// TIA Portal project "LLCCA_PID" (V19)
// LCC Automation AB / (c)Copyright 2024
// Released under the MIT License

(* hardware
DEVICE "LLCCA_PID_HMI"  TP1200 Comfort
   slot 0: "LLCCA_PID_HMI"  TP1200 Comfort  6AV2 124-0MC01-0AX0  17.0.0.0
   slot 1: "HMI_RT_1"  TP1200 Comfort  6AV2 124-0MC01-0AX0  17.0.0.0
   slot 5: "LLCCA_PID_HMI.IE_CP_1"  PROFINET Interface  17.0.0.0
      slot 1: "PROFINET Interface_1"  PROFINET Interface
         slot 1: "Port_1"  Port
         slot 2: "Port_2"  Port
   slot 7: "LLCCA_PID_HMI.MPI/DP_CP_1"  MPI/DP Interface  17.0.0.0
DEVICE "ET 200SP station_1"  ET 200SP-Station
   slot 0: "Rack_0"  Rack  6ES5 710-8MAx1
   slot 1: "LLCCA_PID_PLC"  CPU 1510SP-1 PN  6ES7 510-1DK03-0AB0  V3.1
      slot 32768: "PROFINET interface_1"  X1
         slot 32771: "Port_3"  X1 P3
   slot 2: "Server module_1"  Server module  6ES7 193-6PA00-0AA0  V1.2
      slot 1: "Server module_1"  Server module
   slot 127: "BA 2xRJ45"  BA 2xRJ45  6ES7 193-6AR00-0AA0  V0.0
      slot 32769: "Port_1"  X1 P1  6ES7 193-6AR00-0AA0
      slot 32770: "Port_2"  X1 P2  6ES7 193-6AR00-0AA0
*)

// ===== PLC "LLCCA_PID_PLC"  CPU 1510SP-1 PN =====

DATA_BLOCK "LLCCA_PvSim_LLCCA_PID_DB"   // DB1
{ S7_Optimized_Access := 'TRUE' }
VERSION : 0.1
// stored: InstanceOfName LLCCA_PvSim
"LLCCA_PvSim"
BEGIN
END_DATA_BLOCK

DATA_BLOCK "LLCCA_PID_DB"   // DB2
{ S7_Optimized_Access := 'TRUE' }
AUTHOR : Jacob Holmdahl
VERSION : 0.0
// stored: InstanceOfName LLCCA_PID
"LLCCA_PID"
BEGIN
END_DATA_BLOCK

DATA_BLOCK "LLCCA_PvSim_PID_C_DB"   // DB3
{ S7_Optimized_Access := 'TRUE' }
VERSION : 0.1
// stored: InstanceOfName LLCCA_PvSim
"LLCCA_PvSim"
BEGIN
END_DATA_BLOCK

DATA_BLOCK "RUN_DB"   // DB5
{ S7_Optimized_Access := 'TRUE' }
VERSION : 0.1
// stored: InstanceOfName RUN
"RUN"
BEGIN
END_DATA_BLOCK

DATA_BLOCK "LLCCA_ErrAcc_DB_LLCCA_PID"   // DB10
{ S7_Optimized_Access := 'TRUE' }
VERSION : 0.1
// stored: InstanceOfName LLCCA_ErrAcc
"LLCCA_ErrAcc"
BEGIN
END_DATA_BLOCK

DATA_BLOCK "LLCCA_ErrAcc_DB_PID_C"   // DB11
{ S7_Optimized_Access := 'TRUE' }
VERSION : 0.1
// stored: InstanceOfName LLCCA_ErrAcc
"LLCCA_ErrAcc"
BEGIN
END_DATA_BLOCK

FUNCTION_BLOCK "RUN"   // FB1, FBD
{ S7_Optimized_Access := 'TRUE' }
AUTHOR : Jacob Holmdahl
VERSION : 0.0
   VAR_INPUT
      setpoint : Real;
   END_VAR
   VAR_IN_OUT
      resetAll : Bool;
      resetPvSim : Bool;
      resetPID : Bool;
      resetAccErr : Bool;
   END_VAR
   VAR
      statSetpoint : Real;
   END_VAR
   VAR_TEMP
      tempPv_LCCA_PID : Real;
      tempPv_PID_C : Real;
      tempResetPvSim : Bool;
      tempResetPID : Bool;
      tempResetAccErr : Bool;
   END_VAR
BEGIN

REGION Network 1 (SCL)
   IF #setpoint <> #statSetpoint THEN
     "LLCCA_PID_DB".Setpoint := #setpoint;
     "PID_Compact_1".Setpoint := #setpoint;
     #statSetpoint := #setpoint;
     #resetAccErr := TRUE;
   END_IF;
END_REGION

REGION Network 2
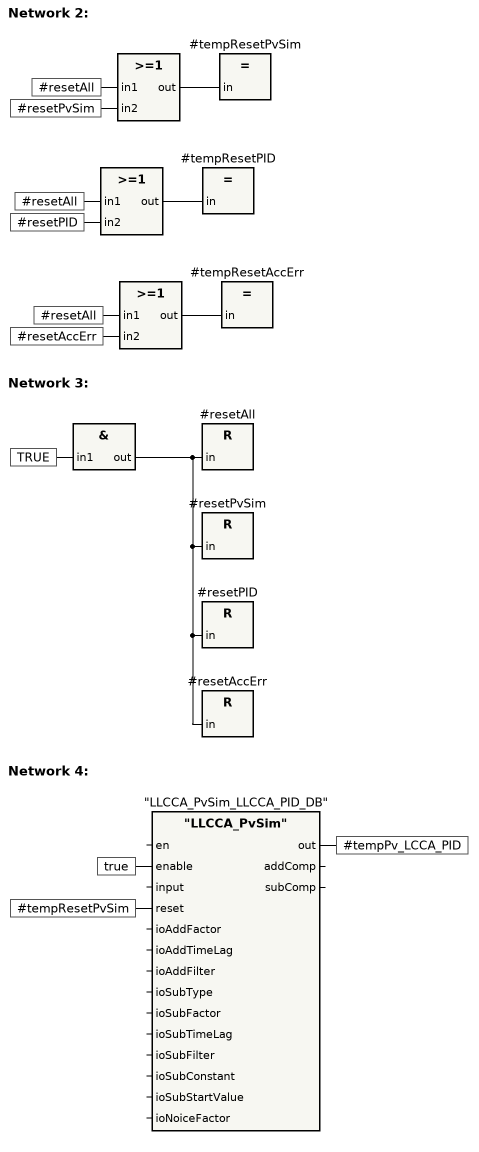
   #tempResetPvSim := #resetAll OR #resetPvSim;
   #tempResetPID := #resetAll OR #resetPID;
   #tempResetAccErr := #resetAll OR #resetAccErr;
END_REGION

REGION Network 3
   IF TRUE THEN
       #resetAll := FALSE;
       #resetPvSim := FALSE;
       #resetPID := FALSE;
       #resetAccErr := FALSE;
   END_IF;
END_REGION

REGION Network 4
   "LLCCA_PvSim_LLCCA_PID_DB"(enable := true, reset := #tempResetPvSim, out => #tempPv_LCCA_PID);   // "LLCCA_PvSim"
END_REGION

REGION Network 5
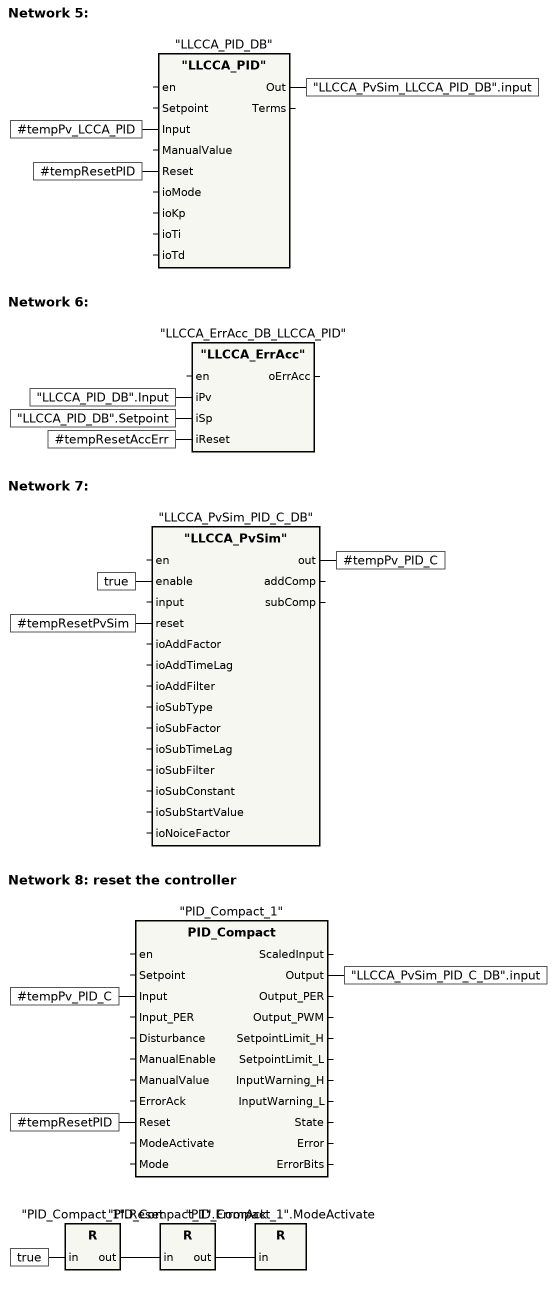
   "LLCCA_PID_DB"(Input := #tempPv_LCCA_PID, Reset := #tempResetPID, Out => "LLCCA_PvSim_LLCCA_PID_DB".input);   // "LLCCA_PID"
END_REGION

REGION Network 6
   "LLCCA_ErrAcc_DB_LLCCA_PID"(iPv := "LLCCA_PID_DB".Input,   // "LLCCA_ErrAcc"
                           iSp := "LLCCA_PID_DB".Setpoint,
                           iReset := #tempResetAccErr);
END_REGION

REGION Network 7
   "LLCCA_PvSim_PID_C_DB"(enable := true, reset := #tempResetPvSim, out => #tempPv_PID_C);   // "LLCCA_PvSim"
END_REGION

REGION Network 8: reset the controller
   "PID_Compact_1"(Input := #tempPv_PID_C, Reset := #tempResetPID, Output => "LLCCA_PvSim_PID_C_DB".input);   // PID_Compact
   IF true THEN
       "PID_Compact_1".Reset := FALSE;
       "PID_Compact_1".ErrorAck := FALSE;
       "PID_Compact_1".ModeActivate := FALSE;
   END_IF;
END_REGION

REGION Network 9
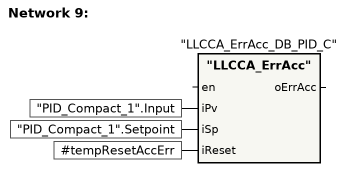
   "LLCCA_ErrAcc_DB_PID_C"(iPv := "PID_Compact_1".Input,   // "LLCCA_ErrAcc"
                           iSp := "PID_Compact_1".Setpoint,
                           iReset := #tempResetAccErr);
END_REGION
END_FUNCTION_BLOCK

FUNCTION_BLOCK "LLCCA_PID"   // FB3, SCL
TITLE = LLCCA_PID
{ S7_Optimized_Access := 'TRUE' }
AUTHOR : Jacob Holmdahl
FAMILY : LLCCA
VERSION : 0.0
// LCC Automation AB / (c)Copyright 2024
// Released under the MIT License
   VAR_INPUT
      Setpoint : Real;   // controller setpoint
      Input : Real;   // current value from the process
      ManualValue : Real;   // manual value
      Reset : Bool;   // reset i term and all filters
   END_VAR
   VAR_OUTPUT
      Out : Real;   // output value
      Terms : Struct   // controller terms
         p : Real;   // proportional term
         i : Real;   // integral term
         d : Real;   // derivative term
      END_STRUCT;
   END_VAR
   VAR_IN_OUT
      ioMode : USInt;   // current mode of operation (0-Inactive, 1-Step tuning, 2-Reserved, 3-Automatic, 4-Manual)
      ioKp : Real := 1.0;   // proportional gain
      ioTi : Real := 3.0;   // integral action time [s]
      ioTd : Real := 0.0;   // derivative action time [s]
   END_VAR
   VAR
      statOut : Real;
   END_VAR
   VAR RETAIN
      statAdvanced : Struct
         outMax : Real := 100.0;   // output value max
         outMin : Real;   // output value min
         inputFilter : Real := 0.1;   // input value filter time [s]
         derivateFilter : Real := 2.0;   // derivative filter time [s]
         tuningRule : USInt;   // 0:CHR 0% 1:0:CHR 20% 11:ZN fast 12:ZN normal 13:ZN slow
      END_STRUCT;
   END_VAR
   VAR
      statStepTuning : Struct
         state : USInt;
         stateInflection : USInt;
         t : Real;   // time
         find_u_max : Real;   // input max
         find_u_min : Real;   // input min
         calc_u_dev : Real;   // input deviation
         calc_u_start : Real;   // input start value
         find_y_start : Real;   // output start value
         find_k_inflection : Real;   // inflection point slope
         find_u_inflection : Real;   // inflection point input
         find_t_inflection : Real;   // inflection point time
         calc_m : Real;   // liniar equation
         calc_dy : Real;   // delta output
         calc_L : Real;   // apparent dead time
         calc_A : Real;
         calc_Kc : Real;
         calc_Ti : Real;
         calc_Td : Real;
      END_STRUCT;
      statErr : Real;
      statRuntime : LReal;
      statIntegralMax : Real;
      statIntegralMin : Real;
      statIntegralSum : Real;
      statMedianFilter : "LLCCA_MedianFilter";
      statFilterPT1 : Filter_PT1;
      "statFilterDT1_du/dt" : Filter_DT1;
      "statFilterDT1_d2u/dt2" : Filter_DT1;
      statMode : USInt;
      statModePrev : USInt;
   END_VAR
   VAR_TEMP
      temp_uM : Real;   // input with median filter
      temp_uF : Real;   // input with PT1 filter
      temp_dt : Real;   // delta time of the controller
      "temp_du/dt" : Real;   // first order derivative
      "temp_d2u/dt2" : Real;   // second order derivative
      temp_out : Real;
   END_VAR
BEGIN
   REGION Header
       //
       //================================================================================== 
       // LCC Automation AB / (c)Copyright 2024
       // Released under the MIT License
       //---------------------------------------------------------------------------------- 
       // Title:            LLCCA_PID
       // Comment/Function: PID Controller with step tuning
       // Library/Family:   LLCCA (Library LCC Automation AB)
       // Author:           Jacob Holmdahl / jacob.holmdahl@lcc.se
       // Target System:    CPU 1510SP-1
       // Engineering:      TIA Portal 19 update 3
       // Restrictions:     none
       // Requirements:     PLC (S7-1200 / S7-1500)
       //---------------------------------------------------------------------------------- 
       // Change log table: 
       // Version     | Date       | Author           | Changes applied
       //-------------|------------|------------------|------------------------------------ 
       // 000.002.000 | 2024-10-22 | Jacob Holmdahl   | PID with integral anti windup
       // 000.003.000 | 2024-11-10 | Jacob Holmdahl   | CHR and ZN step tuning
       // 000.003.001 | 2024-11-27 | Jacob Holmdahl   | First development release
       //==================================================================================
       //
       // Known issues
       // The step tuning only works if the process (input) is very stable.
       // An abort mechanism is needed to stop tuning if the process is or becomes unstable.
       //
       // Information
       // The terminology of some variables and functions is taken from the Siemens PID_Compact
       // controller.
       // 
   END_REGION

   REGION Save previous mode

       // one cycle mode change 
       IF #ioMode <> #statMode THEN
           #statModePrev := #statMode;
           #statMode := #ioMode;

           // init step tuning
           IF #statMode = 1 THEN
               #statStepTuning.state := 0;
               #statStepTuning.stateInflection := 0;
           END_IF;

       END_IF;

   END_REGION

   REGION Delta time
       // calculate the time from previous call = controller cycle time
       #temp_dt := LREAL_TO_REAL(RUNTIME(#statRuntime));
   END_REGION

   REGION Filter and derivatives

       // derivate filter min
       IF #statAdvanced.derivateFilter < 0.1 THEN
           #statAdvanced.derivateFilter := 0.1;
       END_IF;

       // filter setpoints
       #statFilterPT1.Lag := #statAdvanced.inputFilter;
       #"statFilterDT1_du/dt".Lag := #statAdvanced.derivateFilter;
       #"statFilterDT1_d2u/dt2".Lag := #statAdvanced.derivateFilter;

       // input value median filter
       #statMedianFilter(iVal := #Input,
                         iReset := #Reset,
                         oVal => #temp_uM);

       // reset all filters
       IF #Reset THEN
           #statFilterPT1.SubstituteOutput := #Input;
           #"statFilterDT1_du/dt".SubstituteOutput := 0.0;
           #"statFilterDT1_d2u/dt2".SubstituteOutput := 0.0;
       END_IF;

       // input value filter PT1
       #statFilterPT1(Input := #temp_uM,
                      Reset := #Reset,
                      Output => #temp_uF);

       // first order derivative
       // derivate filter DT1
       // returns the slope
       #"statFilterDT1_du/dt"(Input := #temp_uF,
                        Reset := #Reset,
                        Output => #"temp_du/dt");

       // second order derivative
       // derivate filter DT1 of the first derivate filter DT1
       // returns the acceleration of the slope
       #"statFilterDT1_d2u/dt2"(Input := #"temp_du/dt",
                        Reset := #Reset,
                        Output => #"temp_d2u/dt2");

   END_REGION

   REGION Modes

       CASE #statMode OF
           0:  // Inactive
               REGION Inactive
                   #statOut := 0.0;
               END_REGION

           1:  // Step tuning

               // The step tuning is designed to work with a FOPDT process model
               // FOPDT stands for First Order Plus Dead Time
               // First Order: This refers to a system that responds to a change in input with a gradual, exponential approach to a new steady state.
               // Dead Time: This represents a delay between when you make a change to the input and when you see any effect on the output. 

               REGION Step tuning

                   CASE #statStepTuning.state OF
                       0:

                           REGION Initialize tuning

                               // init tuning variables
                               #statStepTuning.find_u_max := #temp_uF;
                               #statStepTuning.find_u_min := #temp_uF;
                               #statStepTuning.calc_u_dev := 0.0;
                               #statStepTuning.calc_u_start := 0.0;
                               #statStepTuning.find_k_inflection := 0.0;
                               #statStepTuning.find_u_inflection := 0.0;
                               #statStepTuning.find_t_inflection := 0.0;
                               #statStepTuning.calc_m := 0.0;
                               #statStepTuning.calc_L := 0.0;
                               #statStepTuning.calc_Kc := 0.0;
                               #statStepTuning.calc_Ti := 0.0;
                               #statStepTuning.calc_Td := 0.0;
                               #statStepTuning.t := 5.0;

                               // transition
                               #statStepTuning.state := 1;

                           END_REGION

                       1:

                           REGION Calculate the standard deviation

                               // find min and max input
                               IF #temp_uF > #statStepTuning.find_u_max THEN
                                   #statStepTuning.find_u_max := #temp_uF;
                               END_IF;
                               IF #temp_uF < #statStepTuning.find_u_min THEN
                                   #statStepTuning.find_u_min := #temp_uF;
                               END_IF;

                               // calculate the standard deviation
                               #statStepTuning.calc_u_dev := #statStepTuning.find_u_max - #statStepTuning.find_u_min;

                               // transition
                               // timer run out / calculate starting point
                               IF #statStepTuning.t <= 0.0 THEN
                                   #statStepTuning.t := 0.0;

                                   // adjust derivate filter to coresponting deviation
                                   #statAdvanced.derivateFilter := #statStepTuning.calc_u_dev * 40.0;
                                   #statAdvanced.derivateFilter := #statStepTuning.calc_u_dev * 40.0;

                                   // save starting point
                                   #statStepTuning.calc_u_start := #statStepTuning.find_u_min + #statStepTuning.calc_u_dev / 2;
                                   #statStepTuning.find_k_inflection := #"temp_du/dt"; // save slope

                                   // save start output
                                   #statStepTuning.find_y_start := #statOut;

                                   // increase output to make a step
                                   #statOut := #statAdvanced.outMax;

                                   // change state
                                   #statStepTuning.state := 2;
                               ELSE
                                   // decrease step timer
                                   #statStepTuning.t := #statStepTuning.t - #temp_dt;
                               END_IF;

                           END_REGION

                       2:

                           REGION Find the point of inflection

                               // terminology
                               // L = Deadtime ( Can also be called τ in some documantations )
                               // T = apparent time constant
                               // y = output

                               // linear equation
                               // u = kt + m ( u=pv , t=time )
                               // k = u2-u1 / t2-t1 = du / dt

                               // finding inflection point = k
                               IF #"temp_du/dt" > #statStepTuning.find_k_inflection THEN
                                   #statStepTuning.find_k_inflection := #"temp_du/dt";
                                   #statStepTuning.find_u_inflection := #temp_uF;
                                   #statStepTuning.find_t_inflection := #statStepTuning.t;
                               END_IF;

                               // calculate m from inflection point
                               // u=kt+m => m=u-kt 
                               #statStepTuning.calc_m := #statStepTuning.find_u_inflection - (#statStepTuning.find_k_inflection * #statStepTuning.find_t_inflection);

                               // calculate L, the "apparent dead time" with u=kt+m => t=u-m/k at the staring level.
                               #statStepTuning.calc_L := (#statStepTuning.calc_u_start - #statStepTuning.calc_m) / #statStepTuning.find_k_inflection;

                               // calculate delta y (delta output)
                               #statStepTuning.calc_dy := #statAdvanced.outMax - #statStepTuning.find_y_start;

                               // A = approximation of KL/T
                               #statStepTuning.calc_A := #statStepTuning.calc_u_start - #statStepTuning.calc_m;

                               // increase timer / tuning time t
                               #statStepTuning.t := #statStepTuning.t + #temp_dt;

                               // start tuning
                               IF #statStepTuning.stateInflection = 0 AND #"statFilterDT1_du/dt".Output > 0.1 THEN
                                   #statStepTuning.stateInflection := 1;
                               END_IF;

                               // end tuning
                               IF #statStepTuning.stateInflection = 1 AND #"statFilterDT1_d2u/dt2".Output < 0.0 THEN
                                   #statStepTuning.stateInflection := 2;
                               END_IF;

                               // transition to "Tuning successful"
                               IF #statStepTuning.stateInflection = 2 THEN
                                   #statStepTuning.state := 3;
                               END_IF;



                               CASE #statAdvanced.tuningRule OF

                                   0: // Chien–Hrones–Reswick - tuning for disturbance rejection - with 0% overshot
                                       #statStepTuning.calc_Kc := (0.95 * #statStepTuning.calc_dy) / #statStepTuning.calc_A;
                                       #statStepTuning.calc_Ti := 2.40 * #statStepTuning.calc_L;
                                       #statStepTuning.calc_Td := 0.42 * #statStepTuning.calc_L;
                                   1: // Chien–Hrones–Reswick - tuning for disturbance rejection - with 20% overshot
                                       #statStepTuning.calc_Kc := (1.20 * #statStepTuning.calc_dy) / #statStepTuning.calc_A;
                                       #statStepTuning.calc_Ti := 2.00 * #statStepTuning.calc_L;
                                       #statStepTuning.calc_Td := 0.42 * #statStepTuning.calc_L;
                                   11:  // Ziegler-Nichols - Fast Performance
                                       #statStepTuning.calc_Kc := (1.20 * #statStepTuning.calc_dy) / #statStepTuning.calc_A;
                                       #statStepTuning.calc_Ti := 2.00 * #statStepTuning.calc_L;
                                       #statStepTuning.calc_Td := 0.50 * #statStepTuning.calc_L;
                                   12:  // Ziegler-Nichols - Normal Performance
                                       #statStepTuning.calc_Kc := (0.53 * #statStepTuning.calc_dy) / #statStepTuning.calc_A;
                                       #statStepTuning.calc_Ti := 4.00 * #statStepTuning.calc_L;
                                       #statStepTuning.calc_Td := 0.80 * #statStepTuning.calc_L;
                                   13:  // Ziegler-Nichols - Slow Performance
                                       #statStepTuning.calc_Kc := (0.32 * #statStepTuning.calc_dy) / #statStepTuning.calc_A;
                                       #statStepTuning.calc_Ti := 4.00 * #statStepTuning.calc_L;
                                       #statStepTuning.calc_Td := 0.80 * #statStepTuning.calc_L;

                                   ELSE  // Statement section ELSE

                                       #statAdvanced.tuningRule := 0;

                               END_CASE;

                           END_REGION


                       3:

                           REGION Tuning successful

                               // set new tuning parameters
                               #ioKp := #statStepTuning.calc_Kc;
                               #ioTi := #statStepTuning.calc_Ti;
                               #ioTd := #statStepTuning.calc_Td;

                               // return to previous mode
                               #ioMode := #statModePrev;

                           END_REGION

                       4:

                           REGION Tuning not successful

                               // return to previous mode
                               #ioMode := #statModePrev;

                           END_REGION

                       ELSE  // error
                           ;
                   END_CASE;

               END_REGION

           2:  // Reserved for future mode
               REGION Reserved for future mode

                   // prohibited mode - inactivate controller
                   #ioMode := 0;

               END_REGION

           3:  // Automatic
               REGION Automatic

                   // error calculation
                   #statErr := #Setpoint - #temp_uF;

                   REGION PID terms

                       // proprtional gain term
                       #Terms.p := #ioKp * #statErr;

                       // derivate term
                       #Terms.d := - #ioKp * #ioTd * #"temp_du/dt";

                       // integral sum
                       #statIntegralSum := #statIntegralSum + ((#statErr * #temp_dt) / #ioTi);

                       // integral reset
                       IF #Reset THEN
                           #statIntegralSum := 0.0;
                       END_IF;

                       REGION Anti-integral windup

                           // integral max and min
                           #statIntegralMax := (#statAdvanced.outMax / #ioKp) - (#Terms.d / #ioKp) - #statErr;
                           #statIntegralMin := (#statAdvanced.outMin / #ioKp) - (#Terms.d / #ioKp) - #statErr;

                           // integral max with positive error
                           IF #statIntegralSum >= #statIntegralMax AND #statErr > 0.0 THEN
                               #statIntegralSum := #statIntegralMax;
                           END_IF;

                           // integral mmin with negative error
                           IF #statIntegralSum <= #statIntegralMin AND #statErr < 0.0 THEN
                               #statIntegralSum := #statIntegralMin;
                           END_IF;
                       END_REGION

                       // integral term
                       IF #ioTi > 0.0 THEN
                           #Terms.i := #ioKp * #statIntegralSum;
                       ELSE
                           #ioTi := 0.0;
                           #Terms.i := 0.0;
                       END_IF;

                   END_REGION

                   REGION Output

                       // calculate temporary output
                       #temp_out := #Terms.p + #Terms.i + #Terms.d;

                       // min and max limit
                       IF #temp_out < #statAdvanced.outMin THEN
                           #temp_out := #statAdvanced.outMin;
                       ELSIF #temp_out > #statAdvanced.outMax THEN
                           #temp_out := #statAdvanced.outMax;
                       END_IF;

                       // set output vaiable
                       #statOut := #temp_out;

                   END_REGION

               END_REGION

           4:  // Manual
               REGION Manual

                   // set manual output
                   #statOut := #ManualValue;

               END_REGION

           ELSE  // prohibited mode - inactivate controller

               #ioMode := 0;

       END_CASE;

   END_REGION

   REGION Output value
       #Out := #statOut;
   END_REGION
END_FUNCTION_BLOCK

FUNCTION_BLOCK "LLCCA_PvSim"   // FB19, SCL
TITLE = LLCCA_PvSim
{ S7_Optimized_Access := 'TRUE' }
AUTHOR : Jacob Holmdahl
FAMILY : LLCCA
VERSION : 0.0
// LCC Automation AB / (c)Copyright 2024
// Released under the MIT License
   VAR_INPUT
      enable : Bool;   // enable simulation
      input : Real;   // input (Output from PID) [%]
      reset : Bool;   // reset
   END_VAR
   VAR_OUTPUT
      out : Real;   // simulated process value [unit]
      addComp : Real;   // additive component [unit/min]
      subComp : Real;   // subtracting component [unit/min]
   END_VAR
   VAR_IN_OUT
      ioAddFactor : Real := 1.0;   // additive component factor ( addComp := input * addFactor ; 100% * 0.01 = 1 unit/min )
      ioAddTimeLag : USInt := 1;   // additive component time lag [s]
      ioAddFilter : Real := 5.0;   // additive component filter [s]
      ioSubType : USInt;   // 0:start val proportial 1:constant
      ioSubFactor : Real := 1.0;   // subtracting component factor ( subComp := ( out - subStartVal ) * subFactor ; sub (120 unit - 20 unit *0.01 = 1 unit/min)
      ioSubTimeLag : USInt;   // subtracting component time lag [s]
      ioSubFilter : Real;   // subtracting component filter [s]
      ioSubConstant : Real := 20.0;   // substracting constant
      ioSubStartValue : Real := 20.0;   // subtracting component start value [unit]
      ioNoiceFactor : Real := 0.1;   // random noice factor of simulated process value
   END_VAR
   VAR
      statOut : Real;
      statRuntimeMem : LReal;
      statAddTimeLag : "LLCCA_TimeLag";
      statAddFilter_PT1 : Filter_PT1;
      statSubTimeLag : "LLCCA_TimeLag";
      statSubFilter_PT1 : Filter_PT1;
   END_VAR
   VAR_TEMP
      tempDeltaTime : LReal;
      tempAdd : Real;
      tempSub : Real;
      tempRndError : Bool;
      tempRndStatus : Word;
      tempRndStatusSub : Word;
   END_VAR
BEGIN
   REGION Description header 
       //================================================================================== 
       // LCC Automation AB / (c)Copyright 2024
       // Released under the MIT License
       //---------------------------------------------------------------------------------- 
       // Title:            LLCCA_PvSim
       // Comment/Function: Process value simulator
       // Library/Family:   LLCCA (Library LCC Automation AB)
       // Author:           Jacob Holmdahl / jacob.holmdahl@lcc.se
       // Target System:    CPU 1510SP-1
       // Engineering:      TIA Portal 19 update 3
       // Restrictions:     none
       // Requirements:     PLC (S7-1200 / S7-1500)
       //---------------------------------------------------------------------------------- 
       // Change log table: 
       // Version     | Date       | Author           | Changes applied
       //-------------|------------|------------------|------------------------------------ 
       // 001.000.000 | 2024-11-27 | Jacob Holmdahl   | First release
       //==================================================================================
   END_REGION

   REGION delta time
       #tempDeltaTime := RUNTIME(#statRuntimeMem);
   END_REGION

   REGION reset

     IF #reset OR NOT #enable THEN
       #statOut := #ioSubStartValue;
   END_IF;

   END_REGION

   REGION limits

     IF #ioAddFilter < 0.00 THEN
       #ioAddFilter := 0.00;
     END_IF;

     IF #ioSubFilter < 0.00 THEN
       #ioSubFilter := 0.00;
     END_IF;

   END_REGION

   REGION add component

     #tempAdd := #input / 1.0;

     IF ENO THEN
         #tempAdd := #input * #ioAddFactor;
     ELSE
       #tempAdd := 0.0;
     END_IF;

   END_REGION

   REGION add timeLag

     #statAddTimeLag(in      := #tempAdd,
                     reset   := #reset,
                     timeLag := #ioAddTimeLag);

   END_REGION

   REGION add filter

     IF #ioAddFilter > 0.01 THEN
       #statAddFilter_PT1.Lag := #ioAddFilter;

       #statAddFilter_PT1(Input            := #statAddTimeLag.out,
                          SubstituteOutput := #statAddTimeLag.out,
                          Reset            := #reset,
                          Output           => #tempAdd);
     ELSE
       #tempAdd := #statAddTimeLag.out;
     END_IF;

     #addComp := #tempAdd;

   END_REGION

   REGION addition

     #statOut := #statOut + ((#tempAdd * LREAL_TO_REAL(#tempDeltaTime)) / 60.0);

   END_REGION

   REGION sub component

     IF #ioSubType = 0 THEN

       #tempSub := (#statOut - #ioSubStartValue) * #ioSubFactor;

     ELSIF #ioSubType = 1 THEN

       IF #statOut > #ioSubStartValue THEN
         #tempSub := #ioSubConstant * #ioSubFactor;
       ELSE
         #statOut := #ioSubStartValue;
       END_IF;

     ELSE
       #ioSubType := 0;
     END_IF;

   END_REGION

   REGION sub timeLag

     #statSubTimeLag(in      := #tempSub,
                     reset   := #reset,
                     timeLag := #ioSubTimeLag);

   END_REGION

   REGION sub filter

     IF #ioSubFilter > 0.01 THEN
       #statSubFilter_PT1.Lag := #ioSubFilter;

       #statSubFilter_PT1(Input            := #statSubTimeLag.out,
                          SubstituteOutput := #statSubTimeLag.out,
                          Reset            := #reset,
                          Output           => #tempSub);
     ELSE
       #tempSub := #statSubTimeLag.out;
     END_IF;

     #subComp := #tempSub;

   END_REGION

   REGION substraction

     #statOut := #statOut - (#tempSub * LREAL_TO_REAL(#tempDeltaTime) / 60.0);

   END_REGION

   REGION output and noice
     #out := #statOut - (0.5 * #ioNoiceFactor) + #ioNoiceFactor * "LGF_Random_Real"(error => #tempRndError, status => #tempRndStatus, subfunctionStatus => #tempRndStatusSub);
   END_REGION
END_FUNCTION_BLOCK

ORGANIZATION_BLOCK "Main"   // OB1, FBD, ProgramCycle
TITLE = "Main Program Sweep (Cycle)"
{ S7_Optimized_Access := 'TRUE' }
VERSION : 0.1
   VAR_INPUT
      Initial_Call : Bool;   // Initial call of this OB
      Remanence : Bool;   // =True, if remanent data are available
   END_VAR
BEGIN

REGION Network 1
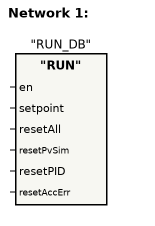
   "RUN_DB"();   // "RUN"
END_REGION
END_ORGANIZATION_BLOCK

// folder: LGF

FUNCTION "LGF_Random_Real" : Real   // FC10077, SCL
TITLE = LGF_Random_Real
{ S7_Optimized_Access := 'TRUE' }
AUTHOR : Siemens_Digital_Industries
FAMILY : LGF
NAME : LGF_Random_Real
// This function generates a random value with each call.  
// The random number has the data type Real in the range from 0.0 to 1.0.
// Diese Funktion generiert bei jedem Aufruf einen zufälligen Wert.  
// Die Zufallszahl hat den Datentyp Real und den Wertebereich von 0.0 bis 1.0.
   VAR_OUTPUT
      error : Bool;   // FALSE: No error TRUE: An error occurred during the execution of the FB / FALSE: Kein Fehler TRUE: Während der Ausführung des FB ist ein Fehler aufgetreten
      status : Word;   // 16#0000-16#7FFF: Status of the FB 16#8000-16#FFFF: Error identification (see following Table) / 16#0000-16#7FFF: Status des FB 16#8000-16#FFFF: Fehleridentifikation (siehe folgende Tabelle)
      subfunctionStatus : Word;   // Status or return value of called FB's, FC's and system blocks / Status oder Rückgabewert von aufgerufenen FB's / FC's und Systemfunktionen
   END_VAR
   VAR_TEMP
      tempTime : DTL;   // Temp memory for System time / Temp variable für System Zeit
      tempNanoSecondInDWord : DWord;   // Temp UDInt converted to DWord for access to individual bytes / Temp UDInt konvertiert nach Dword für den Zufriff per Slice auf die Bytes
      tempTimeStatus : Word;   // Temp status of the instruction `RD_SYS_T` / Temp Status der Systemfunktion `RD_SYS_T`
      tempRandomValue : DWord;   // Temp Random startvalue / Temp Zufallswert als Startwert
   END_VAR
   // Ret_Val : Random Real number between 0.0 and 1.0 / Zufallszahl vom Datentyp Real im Wertebereich von 0.0 bis 1.0
   VAR CONSTANT
      ZERO : Real;   // Zero / 0.0 - value in case of error / Null / 0.0 - Rückgabewert im Fehlerfall
      MAX_UDINT : UDInt := 4294967295 ;   // Maximum UDInt datatype / Maximalwert eines UDInt Datentype
      SUB_STATUS_NO_ERROR : Word := 16#0000;   // Status: sub function call ends without error / Status: Unterfunktionsaufruf ohne Fehler beendet
      STATUS_FINISHED_NO_ERROR : Word := 16#0000;   // Execution finished without errors / Abarbeitung ohne Fehler beendet
      ERR_RD_SYS_T : Word := 16#8600;   // Error in `RD_SYS_T` command - check `subFunctionStatus` code / Fehler in Anweisung `RD_SYS_T` - weitere infos in `subFunctionStatus`
   END_VAR
BEGIN
   REGION Block info header
     //=============================================================================
     // SIEMENS AG / (c)Copyright 2017
     //-----------------------------------------------------------------------------
     // Title:            LGF_Random_Real
     // Comment/Function: Generates a random real number between 0.0 and 1.0
     // Library/Family:   LGF(Library General Functions)
     // Author:           Siemens Digital Industry Support
     // Tested with:      S7-PLCSIM Advanced V2.0 SP1
     // Engineering:      TIA Portal V15 Update 2
     // Restrictions:     ENO disabled - error handling done by error and status
     // Requirements:     PLC (S7-1200 / S7-1500)
     //-------------------------------------------------------------------------------
     // Change log table:
     // Version  | Date       | Expert in charge       | Changes applied
     //----------|------------|------------------------|------------------------------
     // 01.00.00 27.01.2017  Siemens Industry Online Support
     //                      First released version
     // 01.00.01 17.08.2018  Siemens Industry Online Support
     //                      Upgrade: TIA V15 Update 2
     // 01.00.02 23.11.2018  Siemens Industry Online Support
     //                      Upgrade: TIA V15.1
     // 01.01.00 13.11.2019  Simatic Systems Support
     //                      Renamed from "LGF_RandomBasic" to "LGF_Random_Real"
     //                      Regions, comments and constants are added
     // 03.00.00 23.04.2020  Simatic Systems Support
     //                      Set version to V3.0.0, harmonize the version of the whole library
     // 03.00.01 04.02.2021  Simatic Systems Support
     //                      Insert documentation
     //=============================================================================
   END_REGION Block info header

   REGION DESCRIPTION
     (/*Note
   :    The status of called commands is output in `subFunctionStatus`. In this case, the output value in `status` indicates which command caused the error. In this case, refer to the TIA Portal Online Help section for information on the respective commands.

   The function generates random values in the range:  
   $ 0.0 ≤ ReturnVal ≤ 1.0 $.

   The random value is formed from the nanoseconds of the current system time of the CPU. The byte order of this value is inverted and then converted to a floating point.
   Hinweis
   :    In `subFunctionStatus` wird der Status von aufgerufenen Anweisungen ausgegeben. Der Ausgangswert in `status` gibt in diesem Fall an, welche Anweisung den Fehler verursacht hat. Holen Sie sich in diesem Fall die Informationen aus der TIA Portal Online Hilfe zu den jeweiligen Anweisungen.

   Die Funktion generiert zufällige Werte im Bereich:  
   $ 0.0 ≤ ReturnVal ≤ 1.0 $.

   Der Zufallswert wird aus den Nanosekunden der aktuellen Systemzeit der CPU gebildet. Dabei wird die Bytereihenfolge dieses Wertes invertiert und anschließend in eine Gleitkommazahl ungewandelt.*/)
   END_REGION DESCRIPTION

   REGION Validation
     // Read system time
     #tempTimeStatus := INT_TO_WORD(RD_SYS_T(#tempTime));

     // Check return variable for error
     IF (#tempTimeStatus <> #SUB_STATUS_NO_ERROR) THEN
       #error := true;
       #status := #ERR_RD_SYS_T;
       #subfunctionStatus := #tempTimeStatus;
       #LGF_Random_Real := #ZERO;
       RETURN;
     END_IF;
   END_REGION

   REGION Calculating random number
     // Converting to double word so individual bytes can be addressed
     #tempNanoSecondInDWord := UDINT_TO_DWORD(#tempTime.NANOSECOND);

     // Calculate a random-start-value depending on the time
     #tempRandomValue.%B3 := #tempNanoSecondInDWord.%B0;
     #tempRandomValue.%B2 := #tempNanoSecondInDWord.%B1;
     #tempRandomValue.%B1 := #tempNanoSecondInDWord.%B2;
     #tempRandomValue.%B0 := #tempNanoSecondInDWord.%B3;

     // Norm the calculated random number: 0.0 <= Random_Real <= 1.0
     #LGF_Random_Real := UDINT_TO_REAL(DWORD_TO_UDINT(#tempRandomValue)) / UDINT_TO_REAL(#MAX_UDINT);

     #error := false;
     #status := #STATUS_FINISHED_NO_ERROR;
     #subfunctionStatus := #SUB_STATUS_NO_ERROR;
     // ENO mechanism is not used
     ENO := TRUE;
   END_REGION
END_FUNCTION

// folder: SupportFunctions

FUNCTION_BLOCK "LLCCA_ErrAcc"   // FB2, SCL
TITLE = LLCCA_ErrAcc
{ S7_Optimized_Access := 'TRUE' }
AUTHOR : Jacob Holmdahl
FAMILY : LLCCA
VERSION : 0.1
// LCC Automation AB / (c)Copyright 2024
// Released under the MIT License
   VAR_INPUT
      iPv : Real;   // process value
      iSp : Real;   // setpoint
      iReset : Bool;   // reset
   END_VAR
   VAR_OUTPUT
      oErrAcc : LReal;   // error accumulator output
   END_VAR
   VAR
      statErrAcc : LReal;
      statRuntime : LReal;
   END_VAR
   VAR_TEMP
      tempDeltaTime : LReal;
   END_VAR
BEGIN
   REGION Description header 
       //================================================================================== 
       // LCC Automation AB / (c)Copyright 2024
       // Released under the MIT License
       //---------------------------------------------------------------------------------- 
       // Title:            LLCCA_ErrAcc
       // Comment/Function: Process value to setpoint error accumulator
       // Library/Family:   LLCCA (Library LCC Automation AB)
       // Author:           Jacob Holmdahl / jacob.holmdahl@lcc.se
       // Target System:    CPU 1510SP-1
       // Engineering:      TIA Portal 19 update 3
       // Restrictions:     none
       // Requirements:     PLC (S7-1200 / S7-1500)
       //---------------------------------------------------------------------------------- 
       // Change log table: 
       // Version     | Date       | Author           | Changes applied
       //-------------|------------|------------------|------------------------------------ 
       // 001.000.001 | 2024-11-27 | Jacob Holmdahl   | First release
       //==================================================================================
   END_REGION

   #tempDeltaTime := RUNTIME(#statRuntime);

   IF #iReset THEN
       #statErrAcc := 0.0;
   ELSE
       #statErrAcc := #statErrAcc + (ABS(#iSp - #iPv) * #tempDeltaTime);
   END_IF;

   // set output
   #oErrAcc := #statErrAcc;
END_FUNCTION_BLOCK

FUNCTION_BLOCK "LLCCA_MedianFilter"   // FB4, SCL
TITLE = LLCCA_MedianFilter
{ S7_Optimized_Access := 'TRUE' }
AUTHOR : Jacob Holmdahl
FAMILY : LLCCA
VERSION : 0.0
// LCC Automation AB / (c)Copyright 2024
// Released under the MIT License
   VAR_INPUT
      iVal : Real;   // input value
      iReset : Bool;   // reset
   END_VAR
   VAR_OUTPUT
      oVal : Real;   // output value
   END_VAR
   VAR
      statBuffer : Array[0..#UNITS] of Real;
   END_VAR
   VAR_TEMP
      findValue : Real;
      i : Int;
      j : Int;
      tempBuffer : Array[0..#UNITS] of Real;
   END_VAR
   VAR CONSTANT
      UNITS : Int := 31;
   END_VAR
BEGIN
   REGION Description header 
       //================================================================================== 
       // LCC Automation AB / (c)Copyright 2024
       // Released under the MIT License
       //---------------------------------------------------------------------------------- 
       // Title:            LLCCA_MedianFilter
       // Comment/Function: Median filter
       // Library/Family:   LLCCA (Library LCC Automation AB)
       // Author:           Jacob Holmdahl / jacob.holmdahl@lcc.se
       // Target System:    CPU 1510SP-1
       // Engineering:      TIA Portal 19 update 3
       // Restrictions:     none
       // Requirements:     PLC (S7-1200 / S7-1500)
       //---------------------------------------------------------------------------------- 
       // Change log table: 
       // Version     | Date       | Author           | Changes applied
       //-------------|------------|------------------|------------------------------------ 
       // 001.000.000 | 2024-11-27 | Jacob Holmdahl   | First release
       //==================================================================================
   END_REGION

   IF #iReset THEN

       // fill buffer with input val
       FOR #i := 0 TO #UNITS DO
           #statBuffer[#i] := #iVal;
       END_FOR;

       // output is set to input
       #oVal := #iVal;

   ELSE

       // move the static buffer one step
       // and fill the temp buffer
       FOR #i := #UNITS TO 1 BY -1 DO
           #statBuffer[#i] := #statBuffer[#i - 1];
           #tempBuffer[#i] := #statBuffer[#i];
       END_FOR;

       // save the actual value to the buffers
       #statBuffer[0] := #iVal;
       #tempBuffer[0] := #iVal;

       // sort the temp buffer
       FOR #i := 0 TO #UNITS DO
           FOR #j := 0 TO #UNITS - 1 DO
               IF #tempBuffer[#j] > #tempBuffer[#j + 1] THEN
                   #findValue := #tempBuffer[#j];
                   #tempBuffer[#j] := #tempBuffer[#j + 1];
                   #tempBuffer[#j + 1] := #findValue;
               END_IF;
           END_FOR;
       END_FOR;

       // set median val output
       #oVal := (#tempBuffer[#UNITS / 2] + #tempBuffer[#UNITS / 2 + 1]) / 2;

   END_IF;
END_FUNCTION_BLOCK

FUNCTION_BLOCK "LLCCA_TimeLag"   // FB18, SCL
TITLE = LLCCA_TimeLag
{ S7_Optimized_Access := 'TRUE' }
AUTHOR : Jacob Holmdahl
FAMILY : LLCCA
VERSION : 0.0
// LCC Automation AB / (c)Copyright 2024
// Released under the MIT License
   VAR_INPUT
      in : Real;   // input value
      init : Bool;   // time lag memory = in
      reset : Bool;   // time lag memory = 0.0
   END_VAR
   VAR_OUTPUT
      out : Real;   // output value
   END_VAR
   VAR_IN_OUT
      timeLag : USInt := 10;   // time lag [s]
   END_VAR
   VAR
      statRuntimeMem : LReal;
      statTimeLag : Array[0..#TIME_LAG_MAX] of Real;
      statTimer : LReal;
      statInit : Bool;
      statReset : Bool;
   END_VAR
   VAR_TEMP
      tempCycleTime : LReal;
      i : USInt;
   END_VAR
   VAR CONSTANT
      TIME_CYCLE : Real := 0.1;
      TIME_LAG_MAX : USInt := 250;
   END_VAR
BEGIN
   REGION Description header 
       //================================================================================== 
       // LCC Automation AB / (c)Copyright 2024
       // Released under the MIT License
       //---------------------------------------------------------------------------------- 
       // Title:            LLCCA_PID
       // Comment/Function: The output value is delayed by an adjustable time
       // Library/Family:   LLCCA (Library LCC Automation AB)
       // Author:           Jacob Holmdahl / jacob.holmdahl@lcc.se
       // Target System:    CPU 1510SP-1
       // Engineering:      TIA Portal 19 update 3
       // Restrictions:     none
       // Requirements:     PLC (S7-1200 / S7-1500)
       //---------------------------------------------------------------------------------- 
       // Change log table: 
       // Version     | Date       | Author           | Changes applied
       //-------------|------------|------------------|------------------------------------ 
       // 001.000.001 | 2024-11-27 | Jacob Holmdahl   | First release
       //==================================================================================
   END_REGION

   IF #timeLag > 0 THEN

     // run time lag code

     REGION cycleTime
       #tempCycleTime := RUNTIME(#statRuntimeMem);
     END_REGION
     //------------------------------------------------------------------------------------------
     REGION init

       IF #init AND NOT #statInit THEN
         #statInit := TRUE;
         #statTimer := #TIME_CYCLE;
         FOR #i := 0 TO #TIME_LAG_MAX DO
           #statTimeLag[#i] := #in;
         END_FOR;
       ELSIF NOT #init THEN
         #statInit := FALSE;
       END_IF;

     END_REGION
     //------------------------------------------------------------------------------------------
     REGION reset

       IF #reset AND NOT #statReset THEN
         #statReset := TRUE;
         #statTimer := #TIME_CYCLE;
         FOR #i := 0 TO #TIME_LAG_MAX DO
           #statTimeLag[#i] := 0.0;
         END_FOR;
       ELSIF NOT #reset THEN
         #statReset := FALSE;
       END_IF;

     END_REGION
     //------------------------------------------------------------------------------------------
     REGION limits

       // max
       IF #timeLag > #TIME_LAG_MAX/10 THEN
         #timeLag := #TIME_LAG_MAX/10;
       END_IF;

     END_REGION
     //------------------------------------------------------------------------------------------
     // decrease timer
     #statTimer := #statTimer - #tempCycleTime;

     // save value to memory
     IF #statTimer < 0.0 THEN
       #statTimer := #TIME_CYCLE;

       FOR #i := 0 TO #TIME_LAG_MAX-1 DO
         #statTimeLag[#TIME_LAG_MAX - #i] := #statTimeLag[#TIME_LAG_MAX - #i - 1];
       END_FOR;
       #statTimeLag[0] := #in;

     END_IF;

     // set output
     #out := #statTimeLag[#timeLag*10];

   ELSE
     // no time lag

     // set output
     #out := #in;

   END_IF;
END_FUNCTION_BLOCK

// ===== library types =====

// folder: LGF

FUNCTION "LGF_Description" : Void   // FC10087, SCL
TITLE = LGF_Description
{ S7_Optimized_Access := 'TRUE' }
AUTHOR : Siemens Industry Support
NAME : LGF_Description
// Block for the Libray description
BEGIN

   REGION INFO
     (/*title: Library of General Functions (LGF) for SIMATIC S7-1200 / S7-1500
   subTitle: STEP 7 Basic/Professional (TIA PORTAL)
   fileName: LGF
   siosId: 109479728
   link: https://support.industry.siemens.com/cs/ww/en/view/109479728
   classification:   
   # " " "Frei verwendbar" "Unrestricted" "Intern" "Restricted" "Vertraulich" "Confidential" "Streng vertraulich" "Strictly Confidential"
   title: Library of General Functions (LGF) für SIMATIC S7-1200 / S7-1500
   subTitle: STEP 7 Basic/Professional (TIA PORTAL)
   fileName: LGF
   siosId: 109479728
   link: https://support.industry.siemens.com/cs/ww/de/view/109479728
   classification:   
   # " " "Frei verwendbar" "Unrestricted" "Intern" "Restricted" "Vertraulich" "Confidential" "Streng vertraulich" "Strictly Confidential"*/)
   END_REGION INFO

   REGION PREAMBLE
     (/*# Library overview

   ## General information

   TIA Portal has an extensive number of "ready-to-use" instructions (mathematical functions, times, counters, etc.). In addition, there are other useful basic functions.

   These functions are provided in the form of a library and they can be used freely. The finished functions are freely customizable and can therefore be used universally.

   The library described here is versioned and it will be continuously extended. For information on versioning, see Chapter "Versioning".

   ## Hardware and software requirements

   #### Requirements for this library

   In order to be able to use the functionality of the library described here, the following hardware and software requirements must be met.

   #### Hardware

   All blocks (FB, FC, DB, ...) in the library can be used universally with the following controllers:
   * SIMATIC S7-1200 and SIMATIC S7-1200 F product family  
   (from firmware V4.2)
   * SIMATIC S7-1500 and SIMATIC S7-1500 F product family  
   (from firmware V2.0)
   * Simulation with SIMATIC S7-PLCSIM  
   (from V14)

   #### Software

   * SIMATIC STEP 7 Basic/Professional (TIA PORTAL)

   ---

   NOTE
   :    In general, it is possible to open a library with STEP 7 Basic, although STEP 7 Professional elements (e.g. SIMATIC S7-1500 controller) are included. In this case you will be informed with a message when opening the library.
   :    All elements (types and copy templates) can be used if they are supported by the hardware installed in the TIA Portal.
   :    If you try to copy elements with STEP 7 Basic from the library that are not supported (e.g. SIMATIC S7-1500 controller), an error message is displayed.
   # Bibliotheksübersicht

   ## Allgemein

   TIA Portal hat eine umfangreiche Anzahl an "ready-to-use" Anweisungen (Mathematische Funktionen, Zeiten, Zähler, usw.). Darüber hinaus gibt es noch weitere nützliche Basisfunktionen.

   Diese Funktionen werden in Form einer Bibliothek zur Verfügung gestellt und können frei verwendet werden. Die fertigen Funktionen sind frei anpassbar und können somit universell eingesetzt werden.

   Die hier beschriebene Bibliothek ist versioniert und wird kontinuierlich erweitert. Informationen zur Versionierung finden Sie im Anhang Kapitel "Versionierung".

   ## Hard- und Softwarevoraussetzungen

   #### Voraussetzungen für diese Bibliothek

   Um die Funktionalität der hier beschriebenen Bibliothek nutzen zu können, sind nachfolgend genannte Hard- und Softwarevoraussetzungen einzuhalten.

   #### Hardware

   Alle Bausteine (FB, FC, DB, …) in der Bibliothek sind universal mit folgenden Steuerungen einsetzbar:
   * SIMATIC S7-1200 und SIMATIC S7-1200 F Produktfamilie  
   (ab Firmware V4.2)
   * SIMATIC S7-1500 und SIMATIC S7-1500 F Produktfamilie  
   (ab Firmware V2.0)
   * Simulation mit SIMATIC S7-PLCSIM  
   (ab V14)

   #### Software

   * SIMATIC STEP 7 Basic/Professional (TIA PORTAL)

   ---

   Hinweis
   :    Es ist generell möglich eine Bibliothek mit STEP 7 Basic zu öffnen, obwohl STEP 7 Professional Elemente (z.B. SIMATIC S7-1500 Steuerung) enthalten sind. In diesem Fall werden Sie mit einer Meldung beim Öffnen der Bibliothek informiert.   
   :    Es können alle Elemente (Typen und Kopiervorlagen) verwendet werden, wenn sie von der installierten Hardware im TIA Portal unterstützt werden.
   :    Falls Sie versuchen Elemente mit STEP 7 Basic aus der Bibliothek zu kopieren, die nicht unterstützt werden (z.B. SIMATIC S7-1500 Steuerung), wird eine Fehlermeldung angezeigt.*/)

     (/*# Working with the library

   ## General information

   All blocks in the "LGF" library can be used freely in conjunction with SIMATIC S7-1200 and SIMATIC S7-1500 controllers.

   Most of the blocks are stored as types in the library. This means that the blocks are versioned and can thus use all advantages.
   * Central update function for library elements
   * Versioning of library elements

   ---

   Note
   :    Information on the general handling of libraries is provided in the Guideline for Library Handling  
   https://support.industry.siemens.com/cs/ww/en/view/109747503  
   :    and in the Programming Guideline for S7-1200/1500 in the chapter "Libraries".  
   https://support.industry.siemens.com/cs/ww/en/view/81318674

   ---

   Note
   :    All blocks in the LGF were created in accordance with the Programming Style Guide.  
   https://support.industry.siemens.com/cs/ww/en/view/81318674

   ---

   For more information on libraries, visit the TIA Portal:
   * Libraries in the TIA Portal  
     https://support.industry.siemens.com/cs/ww/en/view/109738702

   * How do you open libraries in STEP 7 (TIA Portal)?  
   https://support.industry.siemens.com/cs/ww/en/view/37364723

   * Automate in less than 10 minutes TIA Portal: Time Savers – Global libraries  
     https://support.industry.siemens.com/cs/ww/en/view/78529894

   * Which elements from STEP 7 (TIA Portal) can be stored in a library as a type or as a copy template?  
     https://support.industry.siemens.com/cs/ww/en/view/109476862

   * How can you automatically open a global library when starting TIA Portal V13 or higher and use it e.g. as a corporate library?  
     https://support.industry.siemens.com/cs/ww/en/view/100451450

   * Library with PLC data types for IO module / technology modules and PROFIdrive drives (LPD)  
     https://support.industry.siemens.com/cs/ww/en/view/109482396

   ------

   ## Simulation capability with SIMATIC S7-PLCSIM Advanced

   Simulation with SIMATIC S7-PLCSIM Advanced is already activated in the
   properties of the LGF blocks.

   ![Block properties](LIB_Simulation_01.PNG)

   After translation with SIMATIC S7-PLCSIM Advanced, proceed as follows so that
   the blocks can be simulated.

   1. Open the properties of your project and activate the option "Support simulation during block compilation" in the "Protection" tab.

   ![Project properties](LIB_Simulation_00.PNG)

   ---

   Note
   :    Blocks with activated simulation capability take up more memory space in the PLC.

   ------

   ## User-defined documentation (user help)

   In order to explain the principle of operation and use of the blocks to users of the LGF library, user-defined documentation has been created for each block.  
   The user-defined documentation per block is available in German and English as a PDF file. The PDF files are stored in the following directories of the LGF library.

   * German: `"UserFiles\UserDocumentation\en-DE\Library Types"`
   * English: `"UserFiles\UserDocumentation\en-US\Library Types"`

   The user-defined documentation for a block can be called up in the Task Card "Library" and in the library view with the key combination `<Shift+F1>`.  
   The respective PDF is always opened with the standard program defined in Microsoft Windows.

   So that the user-defined documentation of the blocks can also be called up in the project navigation, you must copy the directories with the PDF files into the project directory `UserFiles`.

   ---

   Note
   :    For user-defined documentation, you require SIMATIC STEP 7 Basic / Professional V15.1 Update 1.

   #### Central directory for user-defined documentation

   Alternatively, you can store the user-defined documentation in a central directory for all projects. To define a central storage location for user help, proceed as follows:

   1. In the "Options" menu, select the "Settings" command.
   2. Open the area "General > General".
   3. Navigate to the "User documentation" section.
   4. Activate the checkbox "Display call log for user-defined documentation" to display a log of the call-up of the user-defined documentation in the Inspector window.
   5. Activate the "Search for user-defined documentation in a central directory" checkbox to store user-defined documentation in a central directory for projects.
   6. In the "Central directory for user-defined documentation" field, specify the path where you want to store cross-project documentation.

   ------

   ![Central directory for user defined documentation](LIB_UserDokumentation.PNG)

   ---

   Note
   :    Do not change the names of the PDF, because the file name must precisely match the name of the object in the TIA Portal.

   ---

   Note
   :    Further information on the user-defined documentation can be found in the system manual "SIMATIC STEP 7 Basic/Professional V15.1 and SIMATIC WinCC V15.1":  
   https://support.industry.siemens.com/cs/ww/en/view/109755202/114872699275
   # Arbeiten mit der Bibliothek

   ## Allgemein

   Alle Bausteine in der Bibliothek "LGF" sind frei verwendbar in Verbindung mit SIMATIC S7-1200 und SIMATIC S7-1500 Steuerungen.

   Der Großteil der Bausteine ist als Typ in der Bibliothek abgelegt. Somit sind die Bausteine versioniert und können somit alle Vorteile nutzen.
   * Zentrale Updatefunktion von Bibliothekselementen
   * Versionierung von Bibliothekselementen

   ---

   Hinweis
   :    Informationen zum generellen Umgang mit Bibliotheken finden Sie im Leitfaden zur Bibliothekshandhabung  
   https://support.industry.siemens.com/cs/ww/de/view/109747503  
   :    und im Programmierleitfaden für S7-1200/1500 im Kapitel "Bibliotheken"  
   https://support.industry.siemens.com/cs/ww/de/view/81318674

   ---

   Hinweis
   :    Alle Bausteine in der LGF wurden nach dem Programmierstyleguide erstellt. https://support.industry.siemens.com/cs/ww/de/view/81318674

   ---

   Weitere Informationen zu Bibliotheken im TIA Portal:
   * Themenseite Bibliotheken  
     https://support.industry.siemens.com/cs/ww/de/view/109738702

   * Wie öffnen Sie Bibliotheken in STEP 7 (TIA Portal)?  
     https://support.industry.siemens.com/cs/ww/de/view/37364723

   * Automatisieren in weniger als 10 Minuten TIA Portal: Time Savers – Globale Bibliotheken  
     https://support.industry.siemens.com/cs/ww/de/view/78529894

   * Welche Elemente aus STEP 7 (TIA Portal) können in einer Bibliothek als Typ oder als Kopiervorlage abgelegt werden?  
     https://support.industry.siemens.com/cs/ww/de/view/109476862

   * Wie können Sie beim Starten von TIA Portal ab V13 eine globale Bibliothek automatisch öffnen und z.B. als Unternehmensbibliothek verwenden?  
     https://support.industry.siemens.com/cs/ww/de/view/100451450

   * Bibliothek mit PLC-Datentypen für Peripherie- / Technologie-Module und PROFIdrive Antriebe (LPD)  
     https://support.industry.siemens.com/cs/ww/de/view/109482396

   ------

   ## Simulierbarkeit mit SIMATIC S7-PLCSIM Advanced

   In den Eigenschaften der LGF Bausteine ist die Simulation mit SIMATIC S7-PLCSIM Advanced bereits aktiviert.

   ![Block properties](LIB_Simulation_01.PNG)

   Damit die Bausteine nach dem Übersetzen mit SIMATIC S7-PLCSIM Advanced
   simuliert werden können, gehen Sie folgendermaßen vor:

   1. Öffnen Sie die Eigenschaften Ihres Projekts und aktivieren Sie im Register "Schutz" die Option "Beim Übersetzen von Bausteinen Simulierbarkeit unterstützen" ("Support simulation during block compilation").

   ![Project properties](LIB_Simulation_00.PNG)

   ---

   Hinweis
   :    Bausteine mit aktivierter Simulierbarkeit belegen mehr Speicherplatz in der PLC.

   ------

   ## Anwenderdefinierte Dokumentation (Anwenderhilfe)

   Um den Anwendern der Bibliothek LGF die Funktionsweise und die Verwendung der Bausteine zu erläutern, wurde für jeden Baustein eine anwenderdefinierte Dokumentation erstellt.  
   Die anwenderdefinierte Dokumentation pro Bausteine ist in den Sprachen Deutsch und Englisch als PDF-Datei verfügbar. Die PDF-Dateien sind in folgenden Verzeichnissen der Bibliothek LGF gespeichert.

   * Deutsch: `"UserFiles\UserDocumentation\de-DE\Library Types"`
   * Englisch: `"UserFiles\UserDocumentation\en-US\Library Types"`

   Die anwenderdefinierte Dokumentation zu einem Baustein können Sie in der Task Card "Bibliothek" und in der Bibliotheksansicht mit der Tastenkombination `<Shift+F1>` aufrufen.  
   Die jeweilige PDF wird immer mit dem in Microsoft Windows festgelegten Standardprogramm geöffnet.

   Damit die anwenderdefinierten Dokumentationen der Bausteine auch in der Projektnavigation aufgerufen werden kann, müssen Sie die Verzeichnisse mit den PDF-Dateien in das Projektverzeichnis "UserFiles" kopieren.

   ---

   Hinweis
   :    Für die Anwenderdefinierte Dokumentation benötigen Sie SIMATIC STEP 7 Basic/Professional V15.1 Update 1.

   #### Zentrales Verzeichnis für anwenderdefinierte Dokumentation

   Alternativ können Sie die anwenderdefinierte Dokumentation auch projektüber-greifend in einem zentralen Verzeichnis ablegen. Um einen zentralen Ablageort für Anwenderhilfe festzulegen, gehen Sie folgendermaßen vor:
   1. Wählen Sie im Menü "Extras" ("Options") den Befehl "Einstellungen" ("Settings").
   2. Öffnen Sie den Bereich "Allgemein > Allgemein" ("General > General").
   3. Navigieren Sie zum Abschnitt "Anwenderdokumentation" ("User documentation").
   4. Aktivieren Sie das Optionskästchen "Aufrufprotokoll zu anwenderdefinierter Dokumentation anzeigen" ("Display call log for user-defined documentation"), um im Inspektor Fenster ein Protokoll vom Aufruf der anwenderdefinierten Dokumentation anzuzeigen.
   5. Aktivieren Sie das Optionskästchen "Suche nach anwenderdefinierter Dokumentation in einem zentralen Verzeichnis" ("Search for user-defined documentation in a central directory"), um anwenderdefinierte Dokumentation in einem projektübergreifenden Verzeichnis abzulegen.
   6. Geben Sie im Feld "Zentrales Verzeichnis für anwenderdefinierte Dokumentation" ("Central directory for user-defined documentation") den Pfad an, an dem Sie projektübergreifende Dokumentation speichern.

   ------

   ![Central directory for user defined documentation](LIB_UserDokumentation.PNG)

   ---

   Hinweis
   :    Ändern Sie nicht die Namen der PDF, denn der Dateiname muss exakt dem
   Namen des Objekts im TIA Portal entsprechen.

   ---

   Hinweis
   :    Weitere Informationen zur anwenderdefinierten Dokumentation finden Sie im
   Systemhandbuch "SIMATIC STEP 7 Basic/Professional V15.1 und SIMATIC
   WinCC V15.1" unter:  
   https://support.industry.siemens.com/cs/ww/de/view/109755202/114872699275*/)

     (/*# Explanation of the blocks

   The chapters below describe all blocks of the library, "Library of General Functions".  
   The chapters have the same structure as the library itself.

   All blocks are divided into application areas or categories:
   * Bit logic operations
   * Date and timer operations
   * Counter operations
   * Comparator operations
   * Math operations
   * Data handling
   * Converter operations
   * Signal generators
   * Technology operations
   * Measurement operations

   ![Global Library (LGF)](LGF_ProjectTree.PNG)
   # Erläuterung der Bausteine

   Die folgenden Kapitel beschreiben alle Bausteine der Bibliothek "Library of General Functions".  
   Die Kapitel sind nach der gleichen Struktur aufgebaut wie die Bibliothek selbst.

   Alle Bausteine sind in Anwendungsgebiete bzw. Kategorien eingeteilt:
   * Bit logic operations (Bitoperationen)
   * Date and timer operations (Datum und Zeitoperationen)
   * Counter operations (Zähloperationen)
   * Comparator operations (Vergleichsoperationen)
   * Math operations (mathematische Operationen)
   * Data handling (Datenverarbeitung)
   * Converter operations (Konvertierungsoperationen)
   * Signal generators (Signalgeneratoren)
   * Technology operations (Technologieoperationen)
   * Measurement operations (Messdatenoperationen)

   ![Global Library (LGF)](LGF_ProjectTree.PNG)*/)
   END_REGION PREAMBLE

   REGION APPENDIX
     (/*# Appendix

   ## Service and support

   #### Industry Online Support
   Do you have any questions or need assistance?  
   Siemens Industry Online Support offers round the clock access to our entire service and support know-how and portfolio.  
   The Industry Online Support is the central address for information about our products, solutions and services.  
   Product information, manuals, downloads, FAQs, application examples and videos, all information is accessible with just a few mouse clicks:  
   https://support.industry.siemens.com

   #### Technical Support
   The Technical Support of Siemens Industry provides you fast and competent support regarding all technical queries with numerous tailor-made offers - ranging from basic support to individual support contracts. Please send queries to Technical Support via Web form:  
   https://www.siemens.com/supportrequest

   #### SITRAIN - Digital Industry Academy
   We support you with our globally available training courses for industry with practical experience, innovative learning methods and a concept that's tailored to the customer's specific needs.  
   For more information on our offered trainings and courses, as well as their locations and dates, refer to our web page:  
   https://www.siemens.com/sitrain

   #### Service offer
   Our range of services includes the following:
   * Plant data services
   * Spare parts services
   * Repair services
   * On-site and maintenance services
   * Retrofitting and modernization services
   * Service programs and contract's

   You can find detailed information on our range of services in the service catalog web page:  
   https://support.industry.siemens.com/cs/sc  

   #### Industry Online Support app
   You will receive optimum support wherever you are with the "Siemens Industry Online Support" app. The app is available for iOS and Android:  
   https://support.industry.siemens.com/cs/ww/en/sc/2067

   ## Industry Mall

   ![Siemens Industry Mall](SiemensIndustryMall.png)

   The Siemens Industry Mall is the platform on which the entire Siemens Industry product portfolio is accessible. From the selection of products to the order and the delivery tracking, the Industry Mall enables the complete purchasing processing – directly and independently of time and location:  
   https://mall.industry.siemens.com
   # Anhang

   ## Service und Support

   #### Industry Online Support
   Sie haben Fragen oder brauchen Unterstützung?  
   Über den Industry Online Support greifen Sie rund um die Uhr auf das gesamte Service und Support Know-how sowie auf unsere Dienstleistungen zu.  
   Der Industry Online Support ist die zentrale Adresse für Informationen zu unseren Produkten, Lösungen und Services.  
   Produktinformationen, Handbücher, Downloads, FAQs und Anwendungsbeispiele, alle Informationen sind mit wenigen Mausklicks erreichbar:  
   https://support.industry.siemens.com

   #### Technical Support
   Der Technical Support von Siemens Industry unterstützt Sie schnell und kompetent bei allen technischen Anfragen mit einer Vielzahl maßgeschneiderter Angebote, von der Basisunterstützung bis hin zu individuellen Supportverträgen.  
   Anfragen an den Technical Support stellen Sie per Web-Formular:  
   https://www.siemens.com/supportrequest

   #### SITRAIN – Digital Industry Academy
   Mit unseren weltweit verfügbaren Trainings für unsere Produkte und Lösungen unterstützen wir Sie praxisnah, mit innovativen Lernmethoden und mit einem kundenspezifisch abgestimmten Konzept.  
   Mehr zu den angebotenen Trainings und Kursen sowie deren Standorte und Termine erfahren Sie unter:  
   https://www.siemens.de/sitrain

   #### Serviceangebot
   Unser Serviceangebot umfasst folgendes:
   * Plant Data Services
   * Ersatzteilservices
   * Reparaturservices
   * Vor-Ort und Instandhaltungsservices
   * Retrofit- und Modernisierungsservices
   * Serviceprogramme und Verträge

   Ausführliche Informationen zu unserem Serviceangebot finden Sie im Servicekatalog:  
   https://support.industry.siemens.com/cs/sc

   #### Industry Online Support App
   Mit der App "Siemens Industry Online Support" erhalten Sie auch unterwegs die optimale Unterstützung. Die App ist für iOS und Android verfügbar:  
   https://support.industry.siemens.com/cs/ww/de/sc/2067

   ## Industry Mall

   ![Siemens Industry Mall](SiemensIndustryMall.png)

   Die Siemens Industry Mall ist die Plattform, auf der das gesamte Produktportfolio von Siemens Industry zugänglich ist. Von der Auswahl der Produkte über die Bestellung und die Lieferverfolgung ermöglicht die Industry Mall die komplette Einkaufsabwicklung – direkt und unabhängig von Zeit und Ort:  
   https://mall.industry.siemens.com*/)


     (/*## Links and Literature
   +-----+-----------------------------------------------------------------------+
   | No. |Topic     
   +=====+=======================================================================+
   | \1\ | Siemens Industry Online Support
   |     | https://support.industry.siemens.com 
   +-----+-----------------------------------------------------------------------+
   | \2\ | Link to the entry page of the application example
   |     | https://support.industry.siemens.com/cs/ww/en/view/109479728
   +-----+-----------------------------------------------------------------------+
   | \3\ | Programming Guidelines and Programming Style guide for SIMATIC S7-1200 and S7-1500
   |     | https://support.industry.siemens.com/cs/ww/en/view/81318674
   +-----+-----------------------------------------------------------------------+
   | \4\ | Library with PLC data types (LPD) for STEP 7 (TIA Portal) and SIMATIC S7-1200 / S7-1500
   |     | https://support.industry.siemens.com/cs/ww/en/view/109482396
   +-----+-----------------------------------------------------------------------+
   | \5\ | Guideline on Library Handling in Tia Portal
   |     | https://support.industry.siemens.com/cs/ww/en/view/109747503
   +-----+-----------------------------------------------------------------------+
   | \6\ | Libraries in the TIA Portal
   |     | https://support.industry.siemens.com/cs/ww/en/view/109738702

   ------
   ## Links und Literatur
   +---------+---------+
   | No.     |Topic     
   +=========+=========+
   | \1\     | Siemens Industry Online Support
   |         | https://support.industry.siemens.com 
   +---------+---------+
   | \2\     | Link auf die Beitragsseite des Anwendungsbeispiels
   |         | https://support.industry.siemens.com/cs/ww/de/view/109479728
   +---------+---------+
   | \3\     | Programmierleitfaden und Programmierstyleguide für SIMATIC S7-1200 and S7-1500
   |         | https://support.industry.siemens.com/cs/ww/de/view/81318674
   +---------+---------+
   | \4\     | Bibliothek mit PLC-Datentypen (LPD) für STEP 7 (TIA Portal) und SIMATIC S7-1200 / S7-1500
   |         | https://support.industry.siemens.com/cs/ww/de/view/109482396
   +---------+---------+
   | \5\     | Leitfaden zur Bibliothekshandhabung
   |         | https://support.industry.siemens.com/cs/ww/de/view/109747503
   +---------+---------+
   | \6\     | Themenseite Bibliotheken
   |         | https://support.industry.siemens.com/cs/ww/de/view/109738702

   ------*/)

     (/*## Change documentation

   #### Versioning of the library
   The library and library elements are maintained in accordance with the table below:

   +----+-------------------------------------------+-----------------------------------------+--------------------+
   | P  | 1.                                        | 2.                                      | 3.                 |
   +====+===========================================+=========================================+====================+
   |    | Non-compatible change                     | Compatible change                       | Error correction   |
   +----+-------------------------------------------+-----------------------------------------+--------------------+
   |    | * Reduction of interfaces                 | * Extension of the interfaces           | * Bug fix          |
   |    | * Changing the interfaces                 | * Compatible extension of functionality |                    |
   |    | * Incompatible extension of functionality |                                         |                    |

   #### Versioning example

   Example for changing the version:  

   | Library | FB1 | FB2 | FC1 | FC2 | Comment |
   | --- | --- | --- | --- | --- | --- |
   | 1.0.0 | 1.0.0 | 1.0.0 | 1.0.0 | - | Released | 
   | 1.0.1 | 1.0.1 | 1.0.0 | 1.0.0 | - | Troubleshooting of FB1 | 
   | 1.0.2 | 1.0.1 | 1.0.1 | 1.0.0 | - | Optimization of FB2 | 
   | 1.1.0 | 1.1.0 | 1.0.1 | 1.0.0 | - | Extension to FB1 | 
   | 1.2.0 | 1.2.0 | 1.0.1 | 1.0.0 | - | Extension to FB1 | 
   | 2.0.0 | 2.0.0 | 1.0.1 | 2.0.0 | - | New functionality on FB1 and FC1 | 
   | 2.0.1 | 2.0.0 | 1.0.2 | 2.0.0 | - | Troubleshooting FB2 | 
   | 3.0.0 | 2.0.0 | 1.0.2 | 2.0.0 | 1.0.0 | New function FC2 | 
   | 3.0.1 | 2.0.1 | 1.0.3 | 2.0.1 | 1.0.1 | Upgrade to new TIA Portal version | 
   | 3.0.2 | 2.0.2 | 1.0.4 | 2.0.2 | 1.0.1 | New functions, bug fixes |
   ## Änderungsdokumentation

   #### Versionierung der Bibliothek
   Die Bibliothek und Bibliothekselemente werden gemäß folgender Tabelle gepflegt:

   +----+-----------------------------------------------+---------------------------------------------+-----------------+
   | P  | 1.                                            | 2.                                          | 3.              |
   +====+===============================================+=============================================+=================+
   |    | Nichtkompatible Änderung                      | Kompatible Änderung                         | Fehlerkorrektur |
   +----+-----------------------------------------------+---------------------------------------------+-----------------+
   |    | * Reduzierung der Schnittstellen              | * Erweiterung der Schnittstellen            | * Bugfix        |
   |    | * Ändern der Schnittstellen                   | * Kompatible Erweiterung der Funktionalität |                 |
   |    | * Inkompatible Erweiterung der Funktionalität |                                             |                 |

   #### Versionierungs Beispiel

   Beispiel für das ändern und hochzählen der Versionsnummer:

   |  Library | FB1 | FB2 | FC1 | FC2 | Comment |
   | --- | --- | --- | --- | --- | --- |
   | 1.0.0 | 1.0.0 | 1.0.0 | 1.0.0 | - | freigegeben | 
   | 1.0.1 | 1.0.1 | 1.0.0 | 1.0.0 | - | Fehlerbehebung von FB1 | 
   | 1.0.2 | 1.0.1 | 1.0.1 | 1.0.0 | - | Optimierung von FB2 | 
   | 1.1.0 | 1.1.0 | 1.0.1 | 1.0.0 | - | Erweiterung an FB1 | 
   | 1.2.0 | 1.2.0 | 1.0.1 | 1.0.0 | - | Erweiterung an FB1 | 
   | 2.0.0 | 2.0.0 | 1.0.1 | 2.0.0 | - | neue Funktionalität an FB1 und FC1 | 
   | 2.0.1 | 2.0.0 | 1.0.2 | 2.0.0 | - | Fehlerbehebung FB2 | 
   | 3.0.0 | 2.0.0 | 1.0.2 | 2.0.0 | 1.0.0 | Neue Funktion FC2 | 
   | 3.0.1 | 2.0.1 | 1.0.3 | 2.0.1 | 1.0.1 | Upgrade auf neue TIA Portal Version | 
   | 3.0.2 | 2.0.2 | 1.0.4 | 2.0.2 | 1.0.1 | Neue Funktionen, Fehlerbehebungen |*/)
   END_REGION APPENDIX
END_FUNCTION

(* ===== HMI "HMI_RT_1" =====
system functions are stored by id; their names below are inferred from use
connection "HMI_Connection_1": ETHERNET, S7_1500_OMS

HMI tags "PID_LCCA"
   "LLCCA_PID_DB_Input" : Real = PLC LLCCA_PID_DB.Input, 100 ms
   "LLCCA_PID_DB_Out" : Real = PLC LLCCA_PID_DB.Out AT %DB1.DBD0, 100 ms
   "LLCCA_PID_DB_Setpoint" : Real = PLC LLCCA_PID_DB.Setpoint AT %DB1.DBD0, 100 ms
   "LLCCA_PID_DB_ioKp" : Real = PLC LLCCA_PID_DB.ioKp AT %DB1.DBX0.0, 1 s
   "LLCCA_PID_DB_ioTi" : Real = PLC LLCCA_PID_DB.ioTi AT %DB1.DBX0.0, 1 s
   "LLCCA_PID_DB_ioTd" : Real = PLC LLCCA_PID_DB.ioTd AT %DB1.DBX0.0, 1 s
   "LLCCA_PID_DB_Terms_p" : Real = PLC LLCCA_PID_DB.Terms.p AT %DB1.DBD0, 100 ms
   "LLCCA_PID_DB_Terms_i" : Real = PLC LLCCA_PID_DB.Terms.i AT %DB1.DBD0, 100 ms
   "LLCCA_PID_DB_Terms_d" : Real = PLC LLCCA_PID_DB.Terms.d AT %DB1.DBD0, 100 ms
   "LLCCA_PID_DB_statIntegralSum" : Real = PLC LLCCA_PID_DB.statIntegralSum AT %DB1.DBD0, 100 ms
   "LLCCA_PID_DB_statAdvanced_outMin" : Real = PLC LLCCA_PID_DB.statAdvanced.outMin AT %DB1.DBD0, 1 s
   "LLCCA_PID_DB_statAdvanced_outMax" : Real = PLC LLCCA_PID_DB.statAdvanced.outMax AT %DB1.DBD0, 1 s
   "LLCCA_PID_DB_statAdvanced_derivateFilter" : Real = PLC LLCCA_PID_DB.statAdvanced.derivateFilter AT %DB1.DBD0, 1 s
   "LLCCA_PID_DB_ioMode" : USInt = PLC LLCCA_PID_DB.ioMode AT %DB1.DBD0, 100 ms
   "LLCCA_PID_DB_ManualValue" : Real = PLC LLCCA_PID_DB.ManualValue AT %DB1.DBB0, 1 s
   "LLCCA_PID_DB_statStepTuning_state" : USInt = PLC LLCCA_PID_DB.statStepTuning.state AT %DB1.DBD0, 100 ms
   "LLCCA_PID_DB_statStepTuning_t" : Real = PLC LLCCA_PID_DB.statStepTuning.t AT %DB1.DBB0, 100 ms
   "LLCCA_PID_DB_statAdvanced_inputFilter" : Real = PLC LLCCA_PID_DB.statAdvanced.inputFilter AT %DB1.DBD0, 1 s
   "LLCCA_PID_DB_statAdvanced_tuningRule" : USInt = PLC LLCCA_PID_DB.statAdvanced.tuningRule AT %DB1.DBD0, 1 s

HMI tags "PID_Compact"
   "PID_Compact_1_Input" : Real = PLC PID_Compact_1.Input AT %DB1.DBD0, 100 ms
   "PID_Compact_1_Output" : Real = PLC PID_Compact_1.Output AT %DB1.DBD0, 100 ms
   "PID_Compact_1_Setpoint" : Real = PLC PID_Compact_1.Setpoint AT %DB1.DBX0.0, 100 ms
   "PID_Compact_1_Input_PER" : Int = PLC PID_Compact_1.Input_PER AT %DB1.DBD0, 1 s
   "PID_Compact_1_Disturbance" : Real = PLC PID_Compact_1.Disturbance AT %DB1.DBD0, 1 s
   "PID_Compact_1_ManualEnable" : Bool = PLC PID_Compact_1.ManualEnable AT %DB1.DBD0, 1 s
   "PID_Compact_1_ManualValue" : Real = PLC PID_Compact_1.ManualValue AT %DB1.DBD0, 1 s
   "PID_Compact_1_ErrorAck" : Bool = PLC PID_Compact_1.ErrorAck AT %DB1.DBD0, 1 s
   "PID_Compact_1_Reset" : Bool = PLC PID_Compact_1.Reset AT %DB1.DBD0, 1 s
   "PID_Compact_1_ModeActivate" : Bool = PLC PID_Compact_1.ModeActivate AT %DB1.DBD0, 1 s
   "PID_Compact_1_ScaledInput" : Real = PLC PID_Compact_1.ScaledInput AT %DB1.DBD0, 1 s
   "PID_Compact_1_Output_PER" : Int = PLC PID_Compact_1.Output_PER AT %DB1.DBD0, 1 s
   "PID_Compact_1_Output_PWM" : Bool = PLC PID_Compact_1.Output_PWM AT %DB1.DBD0, 1 s
   "PID_Compact_1_SetpointLimit_H" : Bool = PLC PID_Compact_1.SetpointLimit_H AT %DB1.DBD0, 1 s
   "PID_Compact_1_SetpointLimit_L" : Bool = PLC PID_Compact_1.SetpointLimit_L AT %DB1.DBD0, 1 s
   "PID_Compact_1_InputWarning_H" : Bool = PLC PID_Compact_1.InputWarning_H AT %DB1.DBD0, 1 s
   "PID_Compact_1_InputWarning_L" : Bool = PLC PID_Compact_1.InputWarning_L AT %DB1.DBD0, 1 s
   "PID_Compact_1_State" : Int = PLC PID_Compact_1.State AT %DB1.DBD0, 1 s
   "PID_Compact_1_Error" : Bool = PLC PID_Compact_1.Error AT %DB1.DBD0, 1 s
   "PID_Compact_1_ErrorBits" : DWord = PLC PID_Compact_1.ErrorBits AT %DB1.DBD0, 1 s
   "PID_Compact_1_Mode" : Int = PLC PID_Compact_1.Mode AT %DB1.DBD0, 1 s
   "PID_Compact_1_InternalVersion" : DWord = PLC PID_Compact_1.InternalVersion AT %DB1.DBD0, 1 s
   "PID_Compact_1_IntegralResetMode" : Int = PLC PID_Compact_1.IntegralResetMode AT %DB1.DBD0, 1 s
   "PID_Compact_1_OverwriteInitialOutputValue" : Real = PLC PID_Compact_1.OverwriteInitialOutputValue AT %DB1.DBD0, 1 s
   "PID_Compact_1_RunModeByStartup" : Bool = PLC PID_Compact_1.RunModeByStartup AT %DB1.DBD0, 1 s
   "PID_Compact_1_LoadBackUp" : Bool = PLC PID_Compact_1.LoadBackUp AT %DB1.DBD0, 1 s
   "PID_Compact_1_SetSubstituteOutput" : Bool = PLC PID_Compact_1.SetSubstituteOutput AT %DB1.DBD0, 1 s
   "PID_Compact_1_PhysicalUnit" : Int = PLC PID_Compact_1.PhysicalUnit AT %DB1.DBD0, 1 s
   "PID_Compact_1_PhysicalQuantity" : Int = PLC PID_Compact_1.PhysicalQuantity AT %DB1.DBD0, 1 s
   "PID_Compact_1_ActivateRecoverMode" : Bool = PLC PID_Compact_1.ActivateRecoverMode AT %DB1.DBD0, 1 s
   "PID_Compact_1_Warning" : DWord = PLC PID_Compact_1.Warning AT %DB1.DBD0, 1 s
   "PID_Compact_1_WarningInternal" : DWord = PLC PID_Compact_1.WarningInternal AT %DB1.DBD0, 1 s
   "PID_Compact_1_Progress" : Real = PLC PID_Compact_1.Progress AT %DB1.DBD0, 1 s
   "PID_Compact_1_CurrentSetpoint" : Real = PLC PID_Compact_1.CurrentSetpoint AT %DB1.DBD0, 1 s
   "PID_Compact_1_CancelTuningLevel" : Real = PLC PID_Compact_1.CancelTuningLevel AT %DB1.DBD0, 1 s
   "PID_Compact_1_SubstituteOutput" : Real = PLC PID_Compact_1.SubstituteOutput AT %DB1.DBD0, 1 s
   "PID_Compact_1_Config" : PID_CompactConfig = PLC PID_Compact_1.Config AT %DB1.DBD0, 1 s
   "PID_Compact_1_CycleTime" : PID_CycleTime = PLC PID_Compact_1.CycleTime AT %DB1.DBD0, 1 s
   "PID_Compact_1_CtrlParamsBackUp" : PID_CompactControlParams = PLC PID_Compact_1.CtrlParamsBackUp AT %DB1.DBD0, 1 s
   "PID_Compact_1_PIDSelfTune" : PID_CompactSelfTune = PLC PID_Compact_1.PIDSelfTune AT %DB1.DBD0, 1 s
   "PID_Compact_1_PIDCtrl" : PID_CompactControl = PLC PID_Compact_1.PIDCtrl AT %DB1.DBD0, 100 ms
   "PID_Compact_1_Retain" : PID_CompactRetain = PLC PID_Compact_1.Retain AT %DB1.DBD0, 1 s

HMI tags "_RUN"
   "RUN_DB_resetAll" : Bool = PLC RUN_DB.resetAll AT %DB1.DBD0, 100 ms
   "RUN_DB_resetPID" : Bool = PLC RUN_DB.resetPID AT %DB1.DBD0, 100 ms
   "RUN_DB_resetPvSim" : Bool = PLC RUN_DB.resetPvSim AT %DB1.DBD0, 100 ms
   "RUN_DB_resetAccErr" : Bool = PLC RUN_DB.resetAccErr AT %DB1.DBX0.0, 1 s
   "RUN_DB_setpoint" : Real = PLC RUN_DB.setpoint AT %DB1.DBX0.0, 1 s

HMI tags "LCCA_PvSim_LCCA_PID"
   "LLCCA_PvSim_LLCCA_PID_DB_enable" : Bool = PLC LLCCA_PvSim_LLCCA_PID_DB.enable, 1 s
   "LLCCA_PvSim_LLCCA_PID_DB_input" : Real = PLC LLCCA_PvSim_LLCCA_PID_DB.input, 100 ms
   "LLCCA_PvSim_LLCCA_PID_DB_out" : Real = PLC LLCCA_PvSim_LLCCA_PID_DB.out, 100 ms
   "LLCCA_PvSim_LLCCA_PID_DB_addComp" : Real = PLC LLCCA_PvSim_LLCCA_PID_DB.addComp, 100 ms
   "LLCCA_PvSim_LLCCA_PID_DB_subComp" : Real = PLC LLCCA_PvSim_LLCCA_PID_DB.subComp, 100 ms
   "LLCCA_PvSim_LLCCA_PID_DB_reset" : Bool = PLC LLCCA_PvSim_LLCCA_PID_DB.reset, 1 s
   "LLCCA_PvSim_LLCCA_PID_DB_ioAddFactor" : Real = PLC LLCCA_PvSim_LLCCA_PID_DB.ioAddFactor, 1 s
   "LLCCA_PvSim_LLCCA_PID_DB_ioAddTimeLag" : USInt = PLC LLCCA_PvSim_LLCCA_PID_DB.ioAddTimeLag, 1 s
   "LLCCA_PvSim_LLCCA_PID_DB_ioAddFilter" : Real = PLC LLCCA_PvSim_LLCCA_PID_DB.ioAddFilter, 1 s
   "LLCCA_PvSim_LLCCA_PID_DB_ioSubFactor" : Real = PLC LLCCA_PvSim_LLCCA_PID_DB.ioSubFactor, 1 s
   "LLCCA_PvSim_LLCCA_PID_DB_ioSubStartValue" : Real = PLC LLCCA_PvSim_LLCCA_PID_DB.ioSubStartValue, 1 s
   "LLCCA_PvSim_LLCCA_PID_DB_ioNoiceFactor" : Real = PLC LLCCA_PvSim_LLCCA_PID_DB.ioNoiceFactor AT %DB1.DBD0, 1 s
   "LLCCA_PvSim_LLCCA_PID_DB_ioSubConstant" : Real = PLC LLCCA_PvSim_LLCCA_PID_DB.ioSubConstant AT %DB1.DBD0, 1 s
   "LLCCA_PvSim_LLCCA_PID_DB_ioSubType" : USInt = PLC LLCCA_PvSim_LLCCA_PID_DB.ioSubType AT %DB1.DBD0, 1 s
   "LLCCA_PvSim_LLCCA_PID_DB_ioSubTimeLag" : USInt = PLC LLCCA_PvSim_LLCCA_PID_DB.ioSubTimeLag AT %DB1.DBB0, 1 s
   "LLCCA_PvSim_LLCCA_PID_DB_ioSubFilter" : Real = PLC LLCCA_PvSim_LLCCA_PID_DB.ioSubFilter AT %DB1.DBB0, 1 s

HMI tags "LCCA_PvSim_PID_C"
   "LLCCA_PvSim_PID_C_DB_enable" : Bool = PLC LLCCA_PvSim_PID_C_DB.enable, 1 s
   "LLCCA_PvSim_PID_C_DB_input" : Real = PLC LLCCA_PvSim_PID_C_DB.input, 100 ms
   "LLCCA_PvSim_PID_C_DB_out" : Real = PLC LLCCA_PvSim_PID_C_DB.out, 100 ms
   "LLCCA_PvSim_PID_C_DB_addComp" : Real = PLC LLCCA_PvSim_PID_C_DB.addComp, 100 ms
   "LLCCA_PvSim_PID_C_DB_subComp" : Real = PLC LLCCA_PvSim_PID_C_DB.subComp, 100 ms
   "LLCCA_PvSim_PID_C_DB_reset" : Bool = PLC LLCCA_PvSim_PID_C_DB.reset, 1 s
   "LLCCA_PvSim_PID_C_DB_ioAddFactor" : Real = PLC LLCCA_PvSim_PID_C_DB.ioAddFactor, 1 s
   "LLCCA_PvSim_PID_C_DB_ioAddTimeLag" : USInt = PLC LLCCA_PvSim_PID_C_DB.ioAddTimeLag, 1 s
   "LLCCA_PvSim_PID_C_DB_ioAddFilter" : Real = PLC LLCCA_PvSim_PID_C_DB.ioAddFilter, 1 s
   "LLCCA_PvSim_PID_C_DB_ioSubFactor" : Real = PLC LLCCA_PvSim_PID_C_DB.ioSubFactor, 1 s
   "LLCCA_PvSim_PID_C_DB_ioSubStartValue" : Real = PLC LLCCA_PvSim_PID_C_DB.ioSubStartValue, 1 s
   "LLCCA_PvSim_PID_C_DB_ioNoiceFactor" : Real = PLC LLCCA_PvSim_PID_C_DB.ioNoiceFactor AT %DB1.DBD0, 1 s
   "LLCCA_PvSim_PID_C_DB_ioSubConstant" : Real = PLC LLCCA_PvSim_PID_C_DB.ioSubConstant AT %DB1.DBD0, 1 s
   "LLCCA_PvSim_PID_C_DB_ioSubType" : USInt = PLC LLCCA_PvSim_PID_C_DB.ioSubType AT %DB1.DBD0, 1 s
   "LLCCA_PvSim_PID_C_DB_ioSubTimeLag" : USInt = PLC LLCCA_PvSim_PID_C_DB.ioSubTimeLag AT %DB1.DBB0, 1 s
   "LLCCA_PvSim_PID_C_DB_ioSubFilter" : Real = PLC LLCCA_PvSim_PID_C_DB.ioSubFilter AT %DB1.DBB0, 1 s

HMI tags "AccError"
   "LLCCA_ErrAcc_DB_LLCCA_PID_oErrAcc" : LReal = PLC LLCCA_ErrAcc_DB_LLCCA_PID.oErrAcc, 100 ms
   "LLCCA_ErrAcc_DB_PID_C_oErrAcc" : LReal = PLC LLCCA_ErrAcc_DB_PID_C.oErrAcc AT %DB1.DBX0.0, 100 ms

text list "PID_C_controller_state_read": 0 'Inactive / Inaktiv'; 1 'Pretuning'; 2 'Fine tuning'; 3 'Auto'; 4 'Manual / Manuell'; 5 'Error / Fel'

text list "PID_C_controller_state_write": 0 'Inactive / Inaktiv'; 1 'Pretuning'; 2 'Fine tuning'; 3 'Auto'; 4 'Manual / Manuell'

text list "PID_C_controller_fine_tuning": 0 'PID automatic'; 1 'PID fast'; 2 'PID slow'; 3 'Ziegler-Nichols PID'; 4 'Ziegler-Nichols PI'; 5 'Ziegler-Nichols P'

text list "PID_C_controller_pretuning": 0 'Chien, Hrones, Reswick PID'; 1 'Chien, Hrones, Reswick PI'

text list "PID_C_controller_error": 0 'no error'; 1 'The "Input" parameter is outside the process value limits'; 2 'Invalid value at "Input_PER" parameter. Check whether an error is pending at the analog input.'; 4 'Error during fine tuning. Oscillation of the process value could not be maintained.'; 8 'Error at start of pretuning. The process value is too close to the setpoint. Start fine tuning.'; 16 'The setpoint was changed during tuning.'; 32 'Pretuning is not permitted during fine tuning.'; 128 'Error during pretuning. The output value limits are not configured correctly or the actual value does not react as expected.'; 256 'Error during fine tuning resulted in invalid parameters.'; 512 'Invalid value at "Input" parameter: Value has an invalid number format.'; 1024 'Calculation of output value failed. Check the PID parameters.'; 2048 'Sampling time error: PID_Compact is not called within the sampling time of the cyclic interrupt OB.'; 4096 'Invalid value at "Setpoint" parameter: Value has an invalid number format.'; 65536 'Invalid value at ManualValue parameter. Value has an invalid number format.'; 131072 'Invalid value at SubstituteOutput tag. Value has an invalid number format.'; 262144 'Invalid value at Disturbance parameter. Value has an invalid number format.'

text list "LLCCA_PID_stepTuning_state": 0 'Initialize tuning'; 1 'Calculate the standard deviation'; 2 'Find the point of inflection'; 3 'Tuning successful'; 4 'Tuning not successful'

text list "LLCCA_PID_stepTuning": 0 'PID Chien, Hrones, Reswick - 0% overshot / Chien, Hrones, Reswick PID'; 1 'PID Chien, Hrones, Reswick - 20% overshot / Chien, Hrones, Reswick PI'; 11 'PID Ziegler-Nichols - Fast Performance / Chien, Hrones, Reswick PI'; 12 'PID Ziegler-Nichols - Normal Performance / Chien, Hrones, Reswick PI'; 13 'PID Ziegler-Nichols - Slow Performance / Chien, Hrones, Reswick PI'

text list "LLCCA_PID_state": 0 'Inactive / Inaktiv'; 1 'Step tuning / Pretuning'; 3 'Auto'; 4 'Manual / Manuell'

screen "_MAIN" 1280x800, template "Template_main"
   TrendView "Trend view_1" at 0,0 size 980x400
   Button "Button_1" at 1030,675 size 131x32; TextOff 'reset pid'
      on Release: SetBit("RUN_DB_resetPID")
   IOField "I/O field_1" at 1014,35 size 71x32; FormatPattern 999.99
      ProcessValue <- "LLCCA_PID_DB_Input"
   IOField "I/O field_2" at 1014,70 size 71x32; FormatPattern 999.9
      ProcessValue <- "LLCCA_PID_DB_Setpoint"
   IOField "I/O field_3" at 1014,105 size 71x32; FormatPattern s999.99
      ProcessValue <- "LLCCA_PID_DB_Out"
   IOField "I/O field_5" at 1014,155 size 71x32; FormatPattern s999.99
      ProcessValue <- "LLCCA_PID_DB_statIntegralSum"
   IOField "I/O field_7" at 1014,325 size 71x32; FormatPattern 999.9
      ProcessValue <- "LLCCA_PID_DB_ioKp"
   IOField "I/O field_8" at 1014,355 size 71x32; FormatPattern 999.9
      ProcessValue <- "LLCCA_PID_DB_ioTi"
   IOField "I/O field_9" at 1014,385 size 71x32; FormatPattern 999.9
      ProcessValue <- "LLCCA_PID_DB_ioTd"
   Button "Button_2" at 1030,630 size 131x32; TextOff 'reset pv sim'
      on Release: SetBit("RUN_DB_resetPvSim")
   TextField "Text field_4" at 985,105 size 30x32; Text 'out'
   TextField "Text field_2" at 985,155 size 30x32; Text 'iS'
   TextField "Text field_5" at 985,35 size 30x32; Text 'pv'
   TextField "Text field_6" at 985,70 size 30x32; Text 'sp'
   TextField "Text field_7" at 985,385 size 30x32; Text 'd'
   TextField "Text field_8" at 985,355 size 30x32; Text 'i'
   TextField "Text field_9" at 985,325 size 30x32; Text 'p'
   IOField "I/O field_10" at 1089,35 size 71x32; FormatPattern 999.99
      ProcessValue <- "PID_Compact_1_Input"
   IOField "I/O field_11" at 1089,70 size 71x32; FormatPattern 999.9
      ProcessValue <- "PID_Compact_1_Setpoint"
   IOField "I/O field_12" at 1089,105 size 71x32; FormatPattern s999.99
      ProcessValue <- "PID_Compact_1_Output"
   IOField "I/O field_13" at 1089,325 size 71x32; FormatPattern 999.9
      ProcessValue <- "Gain"
   IOField "I/O field_14" at 1089,355 size 71x32; FormatPattern 999.9
      ProcessValue <- "Ti"
   IOField "I/O field_15" at 1089,385 size 71x32; FormatPattern 999.9
      ProcessValue <- "Td"
   Button "Button_3" at 1030,755 size 131x32; TextOff 'reset all'
      on Release: SetBit("RUN_DB_resetAll")
   IOField "I/O field_16" at 1089,155 size 71x32; FormatPattern s999.99
      ProcessValue <- "IntegralSum"
   IOField "I/O field_17" at 1014,205 size 71x32; FormatPattern s999.99
      ProcessValue <- "LLCCA_PID_DB_Terms_p"
   IOField "I/O field_18" at 1014,235 size 71x32; FormatPattern s999.99
      ProcessValue <- "LLCCA_PID_DB_Terms_i"
   IOField "I/O field_19" at 1014,265 size 71x32; FormatPattern s999.99
      ProcessValue <- "LLCCA_PID_DB_Terms_d"
   TextField "Text field_10" at 985,265 size 30x32; Text 'd'
   TextField "Text field_11" at 985,235 size 30x32; Text 'i'
   TextField "Text field_12" at 985,205 size 30x32; Text 'p'
   TrendView "Trend view_2" at 0,400 size 980x400
   IOField "I/O field_4" at 1015,465 size 71x32; FormatPattern 99999.9
      ProcessValue <- "LLCCA_ErrAcc_DB_LLCCA_PID_oErrAcc"
   IOField "I/O field_6" at 1090,465 size 71x32; FormatPattern 99999.9
      ProcessValue <- "LLCCA_ErrAcc_DB_PID_C_oErrAcc"
   Button "Button_4" at 1030,715 size 131x32; TextOff 'reset acc error'
      on Release: SetBit("RUN_DB_resetAccErr")
   IOField "I/O field_20" at 1029,590 size 131x32; FormatPattern 999.9
      ProcessValue <- "RUN_DB_setpoint"
   TextField "Text field_1" at 1000,590 size 30x32; Text 'sp'
   TextField "Text field_3" at 1015,435 size 145x32; Text 'accumulated error'
   TextField "Text field_13" at 1030,535 size 130x57; Text 'apply to both for testing and comparing'

screen "SIEMENS_PID_C" 1280x800, template "Template_main"
   TextField "Text field_4" at 10,40 size 49x23; Text 'Mode / Läge'
   SymbolicIOField "Symbolic I/O field_1" at 10,65 size 161x32; TextOn '1'; TextOff '0'; TextList "PID_C_controller_state_write"
      ProcessValue <- "PID_Compact_1_Mode"
   TextField "Text field_12" at 10,105 size 103x23; Text 'Active state / Aktivt läge'
   SymbolicIOField "Symbolic I/O field_2" at 10,130 size 161x32; TextOn '1'; TextOff '0'; TextList "PID_C_controller_state_read"
      ProcessValue <- "PID_Compact_1_State"
   TextField "Text field_14" at 10,270 size 100x23; Text 'Parameters / Parametrar'
   IOField "I/O field_3" at 155,305 size 71x32; Unit  
      ProcessValue <- "Gain"
   IOField "I/O field_5" at 230,305 size 71x32; Unit  
      ProcessValue <- "Ti"
   IOField "I/O field_6" at 305,305 size 71x32; Unit  
      ProcessValue <- "Td"
   IOField "I/O field_7" at 380,305 size 71x32; Unit  
      ProcessValue <- "TdFiltRatio"
   IOField "I/O field_8" at 455,305 size 71x32; Unit  
      ProcessValue <- "PWeighting"
   IOField "I/O field_9" at 530,305 size 71x32; Unit  
      ProcessValue <- "DWeighting"
   IOField "I/O field_10" at 605,305 size 71x32; Unit  
      ProcessValue <- "Cycle"
   TextField "Text field_13" at 155,270 size 15x23; Text 'p'
   TextField "Text field_15" at 230,270 size 10x23; Text 'i'
   TextField "Text field_16" at 305,270 size 15x23; Text 'd'
   TextField "Text field_17" at 380,270 size 41x23; Text 'dFilt'
   TextField "Text field_18" at 455,270 size 73x23; Text 'pWeight'
   TextField "Text field_19" at 530,270 size 73x23; Text 'dWeight'
   TextField "Text field_20" at 605,270 size 47x23; Text 'cycle / cykel'
   IOField "I/O field_18" at 315,130 size 96x32; FormatPattern 999.9; Unit  U 
      ProcessValue <- "PID_Compact_1_Setpoint"
   IOField "I/O field_19" at 435,130 size 96x32; FormatPattern 999.9; Unit  % 
      ProcessValue <- "PID_Compact_1_ManualValue"
   SymbolicIOField "Symbolic I/O field_3" at 10,185 size 1146x32; TextOn '1'; TextOff '0'; TextList "PID_C_controller_error"
      ProcessValue <- "PID_Compact_1_ErrorBits"
   Button "Button_2" at 10,220 size 141x32; TextOff 'Acknowledge / Återställ'
      on Release: SetBit("PID_Compact_1_ErrorAck")
   Button "Button_3" at 195,65 size 96x32; TextOff 'Activate / Aktivera'
      on Release: SetBit("PID_Compact_1_ModeActivate")
   TextField "Text field_2" at 315,105 size 27x23; Text 'Sp / Auto sp'
   TextField "Text field_3" at 435,105 size 75x23; Text 'Man val / Man ut'
   IOField "I/O field_11" at 385,370 size 76x32; FormatPattern 99999; Unit  
      ProcessValue <- "State"
   TextField "Text field_1" at 385,345 size 54x23; Text 'State / Läge'
   IOField "I/O field_12" at 385,435 size 76x32; FormatPattern 99999; Unit  
      ProcessValue <- "State"
   SymbolicIOField "Symbolic I/O field_4" at 10,370 size 361x32; TextOn '1'; TextOff '0'; TextList "PID_C_controller_pretuning"
      ProcessValue <- "TuneRule"
   SymbolicIOField "Symbolic I/O field_5" at 10,435 size 361x32; TextOn '1'; TextOff '0'; TextList "PID_C_controller_fine_tuning"
      ProcessValue <- "TuneRule"
   TextField "Text field_7" at 10,345 size 356x23; Text 'Method for pretuning / start up tuning'
   TextField "Text field_8" at 10,410 size 348x23; Text 'Method for fine tuning / tuning in run'
   TextField "Text field_9" at 385,410 size 54x23; Text 'State / Läge'
   Button "Button_1" at 1170,215 size 106x32; TextOff 'SIE_PID_C / -'
   IOField "I/O field_4" at 220,550 size 66x32; FormatPattern 99.99; Unit  
      ProcessValue <- "LLCCA_PvSim_PID_C_DB_ioAddFactor"
   TextField "Text field_22" at 220,525 size 59x23; Text 'factor / faktor'
   IOField "I/O field_15" at 290,550 size 61x32; FormatPattern 99; Unit  s 
      ProcessValue <- "LLCCA_PvSim_PID_C_DB_ioAddTimeLag"
   TextField "Text field_23" at 290,525 size 45x23; Text 'tLag'
   Button "Button_4" at 220,680 size 156x32; TextOff 'Reset / Återställning'
      on Release: SetBit("RUN_DB_resetPvSim")
   IOField "I/O field_21" at 355,550 size 61x32; FormatPattern 999; Unit  s 
      ProcessValue <- "LLCCA_PvSim_PID_C_DB_ioAddFilter"
   TextField "Text field_25" at 355,525 size 51x23; Text 'filter'
   IOField "I/O field_22" at 220,615 size 66x32; FormatPattern 99.99; Unit  
      ProcessValue <- "LLCCA_PvSim_PID_C_DB_ioSubFactor"
   TextField "Text field_26" at 220,590 size 59x23; Text 'factor / faktor'
   IOField "I/O field_23" at 420,615 size 96x32; FormatPattern 99.9; Unit   U 
      ProcessValue <- "LLCCA_PvSim_PID_C_DB_ioSubStartValue"
   TextField "Text field_27" at 420,590 size 104x23; Text 'start value / omgivningstemp.'
   TextField "Text field_28" at 10,525 size 186x23; Text 'Additive component / Värmning'
   TextField "Text field_29" at 10,590 size 213x23; Text 'subtracting component / Kylning'
   IOField "I/O field_16" at 10,550 size 161x32; FormatPattern 999.9; Unit  U/min 
      ProcessValue <- "LLCCA_PvSim_PID_C_DB_addComp"
   IOField "I/O field_17" at 10,615 size 161x32; FormatPattern 999.9; Unit  U/min 
      ProcessValue <- "LLCCA_PvSim_PID_C_DB_subComp"
   TextField "Text field_30" at 10,655 size 66x23; Text 'Sim Pv / Simulerad temp.'
   IOField "I/O field_24" at 10,680 size 161x32; FormatPattern 999.9; Unit  U 
      ProcessValue <- "LLCCA_PvSim_PID_C_DB_out"
   TextField "Text field_31" at 10,745 size 38x23; Text 'add / värmning'
   TextField "Text field_32" at 5,725 size 107x23; Text 'Calculation / Hur värden beräknas'
   TextField "Text field_33" at 10,765 size 36x23; Text 'sub / kylning'
   TextField "Text field_34" at 95,745 size 325x23; Text '[U/min] = factor * controller out% / [°C/min] = faktor * regulator ut%'
   TextField "Text field_35" at 95,765 size 459x23; Text '[U/min] = factor * (simulated value - start value) / [°C/min] = faktor * (simulerad temp. - omgivningstemp.)'
   IOField "I/O field_1" at 410,680 size 96x32; FormatPattern 9.999; Unit   U 
      ProcessValue <- "LLCCA_PvSim_PID_C_DB_ioNoiceFactor"
   TextField "Text field_5" at 410,655 size 53x23; Text 'noice / omgivningstemp.'
   IOField "I/O field_2" at 850,370 size 96x32; FormatPattern 999; Unit  % 
      ProcessValue <- "PID_Compact_1_Progress"
   TextField "Text field_6" at 850,345 size 67x23; Text 'Tuning'
   IOField "I/O field_20" at 520,615 size 96x32; FormatPattern 99.9; Unit   U 
      ProcessValue <- "LLCCA_PvSim_PID_C_DB_ioSubConstant"
   TextField "Text field_24" at 520,590 size 83x23; Text 'constant / omgivningstemp.'
   IOField "I/O field_25" at 290,615 size 61x32; FormatPattern 99; Unit  s 
      ProcessValue <- "LLCCA_PvSim_PID_C_DB_ioSubTimeLag"
   TextField "Text field_36" at 290,590 size 45x23; Text 'tLag'
   IOField "I/O field_26" at 355,615 size 61x32; FormatPattern 999; Unit  s 
      ProcessValue <- "LLCCA_PvSim_PID_C_DB_ioSubFilter"
   TextField "Text field_37" at 355,590 size 51x23; Text 'filter'
   IOField "I/O field_13" at 555,65 size 96x32; FormatPattern 999; Unit  U 
      ProcessValue <- "PID_Compact_1_Input"
   IOField "I/O field_14" at 675,65 size 96x32; FormatPattern 999; Unit  % 
      ProcessValue <- "PID_Compact_1_Output"
   TextField "Text field_10" at 555,40 size 54x23; Text 'Input / Ärvärde'
   TextField "Text field_11" at 675,40 size 67x23; Text 'Output / Utsignal'
   IOField "I/O field_27" at 555,130 size 96x32; FormatPattern 999; Unit  U 
      ProcessValue <- "PID_Compact_1_Setpoint"
   TextField "Text field_21" at 555,105 size 82x23; Text 'Setpoint / Börvärde'

Template "Template_main" 1280x800
   Button "Template_Button_Main" at 1170,35 size 106x32; TextOff 'Main / Översikt'
      on Release: ActivateScreen("_MAIN", 0)
   Button "Template_Button_4" at 1170,215 size 106x32; TextOff 'SIE_PID_C / -'
      on Release: ActivateScreen("SIEMENS_PID_C", 0)
   Button "Template_Button_5" at 1170,260 size 106x32; TextOff '-'
   Button "Template_Button_6" at 1170,305 size 106x32; TextOff '-'
   Button "Template_Button_7" at 1170,350 size 106x32; TextOff '-'
   DateTimeField "Template_Date/time field_1" at 1005,0 size 266x27
   TextField "Template_Text field_1" at 5,0 size 982x27; Text 'LLCCA Controller vs Siemens PID_Compact / IHP ACS Advanced Control System'
   Button "Template_Button_Back" at 1170,755 size 106x32; TextOff 'Back / Tillbaka'
      on Release: function_efd93a16()
   Button "Template_Button_2" at 1170,125 size 106x32; TextOff 'LLCCA_PID / -'
      on Release: ActivateScreen("LLCCA_PID", 0)
   Button "Template_Button_1" at 1170,80 size 106x32; TextOff '-'
   Button "Template_Button_8" at 1170,395 size 106x32; TextOff '-'
   Button "Template_Button_9" at 1170,440 size 106x32; TextOff '-'
   Button "Template_Button_10" at 1170,485 size 106x32; TextOff '-'
   Button "Template_Button_11" at 1170,530 size 106x32; TextOff '-'
   Button "Template_Button_12" at 1170,575 size 106x32; TextOff '-'
   Button "Template_Button_13" at 1170,620 size 106x32; TextOff '-'
   Button "Template_Button_14" at 1170,665 size 106x32; TextOff '-'
   Button "Template_Button_15" at 1170,710 size 106x32; TextOff 'INFO / -'
      on Release: ActivateScreen("INFO", 0)
   Button "Template_Button_3" at 1169,170 size 106x32; TextOff '-'

